(* CODESYS project SimpleFilterPress

Project tree, tasks and I/O mapping:
  CR1082 : CR1082, ifm electronic, order no. PDM360NG, version 3.3.0.2
    application Application
      libraries: VisuDialogs, * (System); CAA Real Time Clock Extern, * (CAA Technical Workgroup); Standard, 3.5.18.0 (System)
      task Task_30ms (cyclic, interval 30 ms, priority 0) calls IO_Block_Organize, POU_MANUAL_CONTROL
      task VISU_TASK (cyclic, interval t#20ms, priority 15) calls VisuElems.Visu_Prg
      GlobalVariables/
        global variables GVL
        global variables GVL_KeyList
        global variables GVL_KeyList_FT
        global variables GVL_KeyList_RT
        global variables GVL_Program_Variables
      image pool ImagePool
      IO Blocks/
        AL1342 Master block/
          program AL1342_IO_Link_Master_A [ST]
        Input Block/
        data type IO_link_port
        Output block/
      Main/
        visualisation Graph
        visualisation Main_Screen
        visualisation Manual
        visualisation Setpoints
        visualisation Stats
      Pressure_Feed/
        program pressure_transducer_1 [ST]: analog_warnings_action
        visualisation W77_1
        visualisation W78_1
        visualisation W79_1
      Pressure_Hydraulic/
        program pressure_transducer [ST]
        visualisation W77
        visualisation W78
        visualisation W79
      PROGRAM_ROUTINES/
        program IO_Block_Organize [CFC]
        program POU_aSeq_Master [LD]
        program POU_MANUAL_CONTROL [LD]
      global variables pVars
      Sentronic/
        program Feed_Diaphram_Pump [ST]
        program POU_Sentronic_ST [ST]
      program SystemTime [ST]
      Warning system/
        function block create_warning [ST]
        Status light/
        program visu_context [ST]
        visualisation W171
        visualisation W172
        visualisation W25
        visualisation W97
        data type warning_message
        global variables warnings_globals
    Communication : Communication, ifm electronic, version 3.3.0.2
      CAN : CAN, ifm electronic, version 3.3.0.2
      Ethernet : Ethernet, ifm electronic, version 3.3.0.2
    Ethernet_1 : Ethernet, CODESYS, version 4.2.0.0
        settings: IPAddress = [192,168,1,247]; SubnetMask = [255,255,255,0]; GatewayAddress = [192,168,1,1]; MACAddress = [16#00,16#02,16#01,16#7B,16#36,16#8D]; NetworkInterfaceName = 'eth0'; NetworkInterfaceName = "eth0"; SaveCommunicationSettings = FALSE
      Modbus_TCP_Master : Modbus TCP Master, 3S - Smart Software Solutions GmbH, version 4.3.0.0
          settings: AutoReconnect = TRUE
    HMI : HMI, ifm electronic, version 3.3.0.2
      Buzzer : Buzzer, ifm electronic, version 3.3.0.2
          output uiBuzzerFreq : UINT  // Frequency
          output xBuzzerON : BIT  // Buzzer ON
      KeyBoards : KeyBoards, ifm electronic, version 3.3.0.2
        Key_Backlight_settings : Key Backlight settings, ifm electronic, version 3.3.0.2
            output xNightModeON : BIT  // Night Mode ON
        Key_Mapping : Key Mapping, ifm electronic, version 3.3.0.2
        Keys : Keys, ifm electronic, version 3.3.0.2
          LEDs_Keyboard_1 : LEDs Keyboard 1, ifm electronic, version 3.3.0.2
              output LEDsKeyboard1 : WORD  // LEDsKeyboard1
          LEDs_Keyboard_3 : LEDs Keyboard 3, ifm electronic, version 3.3.0.2
              output LEDsKeyboard3 : WORD  // LEDs Keyboard 3
      LCD_Backlight : LCD Backlight, ifm electronic, version 3.3.0.2
          output uiBacklightBrightness : UINT  // Brightness
      User_LEDs : User_LEDs, ifm electronic, version 3.3.0.2
          output LED0 : LED_IEC_A_OUTPUT_MAPPING_TYPE  // User LED 0
    Local_IO : Local IO, ifm electronic, version 3.3.0.2
      Inputs : Inputs, ifm electronic, version 3.3.0.2
          input  IN0000 : IN_MULTIFUNCTION_B_INPUT_MAPPING_TYPE  // IN0000
      Outputs : Outputs, ifm electronic, version 3.3.0.2
          output OUT0000 : OUT_DIGITAL_A_OUTPUT_MAPPING_TYPE  // OUT0000
      System_Inputs : System_Inputs, ifm electronic, version 3.3.0.2
          input  uiVoltageVBB30 : UINT  // Voltage VBB30
          input  uiVoltageVBB15 : UINT  // Voltage VBB15
          input  iTemperature0 : INT  // Board Temperature 0
          input  iTemperature1 : INT  // Board Temperature 1
          input  uiLightSensor : UINT  // Light Sensor
    System_Info : System_Info, ifm electronic, version 3.3.0.2
  ecomatDisplay43inch_64bit : ecomatDisplay43inch_64bit, ifm electronic, order no. 
      , version 3.5.19.4
    application Application
      task VISU_TASK (cyclic, interval 100 ms, priority 31) calls VisuElems.Visu_Prg
      GlobalVariables/
      Main_Task/
      Pressure_Feed/
        program pressure_transducer_1 [ST]
        visualisation W77_1
        visualisation W78_1
      Screens/
      Sentronic/
        program Feed_Diaphram_Pump [ST]
        program POU_Sentronic_ST [ST]
    Communication : Communication, ifm electronic, version 3.5.19.4
      CAN : CAN, ifm electronic, version 3.5.19.4
      Ethernet : Ethernet, ifm electronic, version 3.5.19.4
  5ce3da45-db07-42e7-a21c-a00fff4ed8f6|C:\FCW\Full Circle Water\Controls - Documents\Software Versions\graphics\240px-Info_icon_002.svg.png
  5ce3da45-db07-42e7-a21c-a00fff4ed8f6|C:\FCW\Full Circle Water\Controls - Documents\Software Versions\graphics\AL1342.png
  5ce3da45-db07-42e7-a21c-a00fff4ed8f6|C:\FCW\Full Circle Water\Controls - Documents\Software Versions\graphics\AL1342big.jpg
  5ce3da45-db07-42e7-a21c-a00fff4ed8f6|C:\FCW\Full Circle Water\Controls - Documents\Software Versions\graphics\AL1342closeup.png
  5ce3da45-db07-42e7-a21c-a00fff4ed8f6|C:\FCW\Full Circle Water\Controls - Documents\Software Versions\graphics\AL1940.jpg
  5ce3da45-db07-42e7-a21c-a00fff4ed8f6|C:\FCW\Full Circle Water\Controls - Documents\Software Versions\graphics\AL2330.jpg
  5ce3da45-db07-42e7-a21c-a00fff4ed8f6|C:\FCW\Full Circle Water\Controls - Documents\Software Versions\graphics\AL2341.jpg
  5ce3da45-db07-42e7-a21c-a00fff4ed8f6|C:\FCW\Full Circle Water\Controls - Documents\Software Versions\graphics\alert_icon.png
  5ce3da45-db07-42e7-a21c-a00fff4ed8f6|C:\FCW\Full Circle Water\Controls - Documents\Software Versions\graphics\e_stop_button.png
  5ce3da45-db07-42e7-a21c-a00fff4ed8f6|C:\FCW\Full Circle Water\Controls - Documents\Software Versions\graphics\green_check.png
  5ce3da45-db07-42e7-a21c-a00fff4ed8f6|C:\FCW\Full Circle Water\Controls - Documents\Software Versions\graphics\jescochemtanksmall.png
  5ce3da45-db07-42e7-a21c-a00fff4ed8f6|C:\Users\Joe Elvendahl\Pictures\purgepicture.png
  5ce3da45-db07-42e7-a21c-a00fff4ed8f6|C:\Users\Nathan\Full Circle Water\Controls - Documents\Software Versions\graphics\bluebackground 1280x800.png
  5ce3da45-db07-42e7-a21c-a00fff4ed8f6|C:\Users\Nathan\Full Circle Water\Controls - Documents\Software Versions\graphics\FCW1100.png
  5ce3da45-db07-42e7-a21c-a00fff4ed8f6|C:\Users\Nathan\Full Circle Water\Controls - Documents\Software Versions\graphics\FCW720.png
  5ce3da45-db07-42e7-a21c-a00fff4ed8f6|C:\Users\Nathan\Full Circle Water\Controls - Documents\Software Versions\graphics\Stone Phix.png
  5ce3da45-db07-42e7-a21c-a00fff4ed8f6|C:\Users\Nathan\Full Circle Water\Marketing and Sales - Documents\FCW LOGO and BRANDING\Logo\FCW-Logo_Finals\Logo Finals\Full Circle Logo Final-02.png
  5ce3da45-db07-42e7-a21c-a00fff4ed8f6|graphics\AL2240.png
  5ce3da45-db07-42e7-a21c-a00fff4ed8f6|graphics\AL2400.png
  5ce3da45-db07-42e7-a21c-a00fff4ed8f6|graphics\blowdown_valve.png
  5ce3da45-db07-42e7-a21c-a00fff4ed8f6|graphics\bredel_pump.png
  5ce3da45-db07-42e7-a21c-a00fff4ed8f6|graphics\cone.png
  5ce3da45-db07-42e7-a21c-a00fff4ed8f6|graphics\core_blow_valve.png
  5ce3da45-db07-42e7-a21c-a00fff4ed8f6|graphics\doors_closed.png
  5ce3da45-db07-42e7-a21c-a00fff4ed8f6|graphics\doors_open.png
  5ce3da45-db07-42e7-a21c-a00fff4ed8f6|graphics\doors_partly_open.png
  5ce3da45-db07-42e7-a21c-a00fff4ed8f6|graphics\head_valves.png
  5ce3da45-db07-42e7-a21c-a00fff4ed8f6|graphics\hydraulic_pressure_sensor.png
  5ce3da45-db07-42e7-a21c-a00fff4ed8f6|graphics\hydraulic_pump_contactor.png
  5ce3da45-db07-42e7-a21c-a00fff4ed8f6|graphics\hydraulic_temp_and_level.png
  5ce3da45-db07-42e7-a21c-a00fff4ed8f6|graphics\membrane_squeeze_contactor.png
  5ce3da45-db07-42e7-a21c-a00fff4ed8f6|graphics\metal_aro_pump.jpg
  5ce3da45-db07-42e7-a21c-a00fff4ed8f6|graphics\mixer.png
  5ce3da45-db07-42e7-a21c-a00fff4ed8f6|graphics\plate_shifter.png
  5ce3da45-db07-42e7-a21c-a00fff4ed8f6|graphics\press_open.png
  5ce3da45-db07-42e7-a21c-a00fff4ed8f6|graphics\press_side_view.png
  5ce3da45-db07-42e7-a21c-a00fff4ed8f6|graphics\R08_andR09_masters.jpg
  5ce3da45-db07-42e7-a21c-a00fff4ed8f6|graphics\radar_pod.png
  5ce3da45-db07-42e7-a21c-a00fff4ed8f6|graphics\servo_drives.png
  5ce3da45-db07-42e7-a21c-a00fff4ed8f6|graphics\single_filter_plate.png
  5ce3da45-db07-42e7-a21c-a00fff4ed8f6|graphics\squeeze_transducer.png
  5ce3da45-db07-42e7-a21c-a00fff4ed8f6|graphics\squeeze_valve.png
  5ce3da45-db07-42e7-a21c-a00fff4ed8f6|graphics\vector_hose_pump.jpg
  5ce3da45-db07-42e7-a21c-a00fff4ed8f6|graphics\wet_end_master.png
  text list GlobalTextList
*)

// CR1082/Application/IO Blocks/IO_link_port
TYPE IO_link_port :
	STRUCT 
		vendor_ID: UINT;						//  The vendor ID reported by an IO-Link device.
		device_ID: UINT;						//  The model ID number reported by an IO-Link device.
		
		port_ID: STRING;					//  A text description of the port, ie. 'X.02'.   Used for warning visus, such as 'short circuit on port xx'
		port_number: INT;					//  The simple port number.   Used by modbus libraries to directly read/write if they choose to do so.
		block_name: STRING;					//  The name of the device, ie. 'AL1342'.  Used by visus to describe where something is connected, but also by the modbus libraries for direct reads/writes.
		
		DI_pin_4: BOOL;						//  Digital input #1 (pin 4), if port is configured as an input.
		DI_pin_2: BOOL;						//  Digital input #2 (pin 2).   This pin works if the port is configured as IO-Link or as an input.
		
		not_connected: BOOL;				//  Nothing is connected to the port (only works in IO-Link mode.)
		data_invalid: BOOL;					//  Something is connected but it's not communicating correctly (only works in IO-Link mode.)
		
		short_circuit: BOOL;				//  The device on this port has drawn more current than the port can provide.  (300 mA on an AL1342.)
		
		master_disconnected: BOOL;			//  The master block itself isn't connected, so we should ignore individual device disconnections.
		
		read_word_0: WORD;					//  Process data word 0
		read_word_1: WORD;					//  Process data word 1
		read_word_2: WORD;					//  Process data word 2
		read_word_3: WORD;					//  Process data word 3
		read_word_4: WORD;					//  Process data word 4
		read_word_5: WORD;					//  Process data word 5
		read_word_6: WORD;					//  Process data word 6

		write_word_0: WORD;					//  Write to device word 0
		write_word_1: WORD;					//  Write to device word 1
		write_word_2: WORD;					//  Write to device word 2
		write_word_3: WORD;					//  Write to device word 3
		
		DO_pin_4: BOOL;						//  Set pin 4 to on or off (if the IO-Link port is configured as an output.)
		
	END_STRUCT
END_TYPE

// CR1082/Application/Warning system/warning_message
TYPE warning_message :
	STRUCT 
		detail_warning_visu: STRING := ''; 		//  The exact name of the associated warning visualization.  The warning system uses this string to match visualizations and to match duplicate or fixed messages.
		red: BOOL := FALSE;    					//  Is it a 'red' warning?  (System needs immediate attention.)
		yellow: BOOL := FALSE;   				//  Is it a 'yellow'? warning?  (System needs attention eventually.)
		fixed: BOOL := FALSE;    				//  Has the problem been fixed?
		informational: BOOL := FALSE; 			//  Is this just a general message, not a fault?
		pop_up_everywhere: BOOL := FALSE;  		//  Set if we should immediately switch to the detail warning screen no matter what (high priority.)
		pop_up_contextual: BOOL := FALSE;  		//  Set if we should switch to warning detail screen when they enter the corresponding section of the interface, ie. a VFD fault pops when they go to Return Pump
		contextual_visu: STRING := '';  		//  the visualization we should pop up the warning on.
		short_Description: STRING;   			//  This is the description that will appear in the Warning log.
		audible_alarm: BOOL;     				//  If checked, I suggest adding a 'silence alarm' button to the corresponding Warning visu that sets GVL.siren := FALSE;  Siren automatically silences when you go to a Warnings screen
		time_stamp:	DATE_AND_TIME;   			//  The warning automatically gets time stamped; you never need to set this.
		fixed_date_time: DATE_AND_TIME;			//  When was the message marked as fixed?  Also automatically time-stamped.
		truncated_code: INT;					//  Used to reduce the visualization name to an integer that can be easily passed through say a modbus register.  Automatically generated.
	END_STRUCT
END_TYPE

//  To use these Warning messages, they are either passed to the Warnings() function directly, or assigned to an instance of the create_warning function block (which then sends it as needed
//  to the Warnings() function.)

//  The minimum required fields for a Warning message are:   short_Description, detail_warning_visu, and one of the 'type' flags (red, yellow, fixed, or informational.)
//  Everything else is optional.   Time stamping happens automatically.

//  The tradition (but not requirement) is to set the pop_up_everywhere flag to TRUE for 'red' warnings.

//  Example of a minimal complete Warning message:

//  shorted_port_message: warning := (red := TRUE, detail_warning_visu := 'W276', short_Description := 'Shorted output block port');

// CR1082/Application/pVars
{attribute 'qualified_only'}
VAR_GLOBAL PERSISTENT RETAIN

	run: BOOL; 			// The master enable switch for the system, tied to the button in the upper left corner of the main screen.

	
//  System options

	screen_brightness : USINT := 70; 	// 0-100% screen brightness
	use_metric_units : BOOL; 			// If true, display metric units of measurement
	user_pin: INT := 12345; 			// The system pin number.
	relock_after_x_minutes: TIME:= T#10M;	//  How long should a login with the PIN be good for?
	require_pin_to_change_setting: BOOL := FALSE;
	require_pin_to_start : BOOL := FALSE;
	
	power_restored_time: DATE_AND_TIME;				// The time the system last booted up
	power_lost: DATE_AND_TIME;						// The time we lost power at.
	we_had_power_now: DATE_AND_TIME;				// Tracks the time of the most recent execution of the Status_Light program.

//   Clarifier

gallons_since_last_purge: REAL;
purge_frequency_gallons: INT := 3000;
purge_duration: TIME := T#15S;


//   Flow meter

flow_sensor_pipe_cross_section: REAL;				// The cross section (in square inches) of the pipe the thermal mass flow sensor (SM8621) is installed in.

//  Chemical system

analog_coagulant_sensor_installed: BOOL;			// TRUE if we are using an IO-Link analog level sensor on the coagulant tank.
coagulant_tank_empty_level_inches: INT;				//
coagulant_tank_gallons_per_inch: REAL;				//
coagulant_tank_low_level_warning_inches: INT;		//

analog_floc_concentrate_sensor_installed: BOOL;		// TRUE if we are using an IO-Link analog level sensor on the flocculant concentrate tank.
floc_concentrate_empty_level_inches: INT;
floc_conc_gallons_per_inch: REAL;
floc_conc_low_level_warning_inches: INT;

diluted_floc_analog_sensor_installed: BOOL;			// TRUE if we are using an IO-Link analog level sensor on the flocculant concentrate tank.
diluted_floc_empty_level_inches: INT;
diluted_floc_gallons_per_inch: REAL;
diluted_floc_low_level_warning_inches: INT;

//  Mechanical pit mixer

	mechanical_mixer_installed: BOOL;			//  True if the system has a mechanical pit mixer
	Feed_Diaphram_Pump_Enabled: BOOL;				//  True if the mechanical pit mixer is enabled
	Feed_Pump_Speed: REAL;				//  A percentage speed (100 = max speed, or 60 Hz.)

//  Warning system

	myWarnings: ARRAY [1..16] OF warning_message;
	redWarningPresent: BOOL;					// TRUE if there's an active red (critical) warning
	yellowWarningPresent: BOOL;					// TRUE if there's an active yellow (caution/attention) warning
	blueWarningPresent: BOOL;					// TRUE if there's an active blue (informational) warning
	warningButtonLights: INT;					// Used by the old CR1082 controller to turn on/off button lights for the Warnings screen
	
	slave_trip_code: INT;						// The last fault code generated by the slave plate shifter servo
	master_trip_code: INT;						// The last fault code generated by the master plate shifter servo

	last_warning_number: int;					//  The numerical portion of the warning short code, ie. W-201 becomes '201'.
	
// Water tank
	max_level_inches: REAL := 65;		
	low_level_percent: REAL;
	out_of_water_level_percent: REAL;
	
	// Filter Press Setpoints
		Hydraulic_PSI_Setpoint: REAL;
		Air_Blow_Minutes: REAL;
		Cake_Feed_PSI_Setpoint: REAL;
		Cake_Feed_Time_Delay_Secs: REAL;
		Cake_Stepup_Factor: REAL;
		Sentronic_Word: WORD;
		Sentronic_Real: REAL;
		
		
	
	
//  Pressure transducer

	pressure_transducer_type: INT;			//  The deviceID of the last known pressure transducer we saw from the 'pressure_transducer' program.
	


END_VAR

// CR1082/Application/GlobalVariables/GVL
{attribute 'qualified_only'}
VAR_GLOBAL
	

	runGreenHalo: BOOL := FALSE;  // shows (FALSE) or hides (TRUE) the green 'RUNNING' ring around the RUN/STOP button on the main screen.
	phYellowHalo: BOOL := FALSE;  // TRUE to show a yellow (minor fault) halo around the "pH Control" button on the main screen when there is a minor problem with the pH system
	phRedHalo: BOOL := FALSE;	  // TRUE to show a red (critical fault) halo around the "pH Control" button on the main screen when there is a serious problem with the pH system
	sanitizerYellowHalo: BOOL := TRUE;  // FALSE to show a yellow (minor fault) halo around the "Sanitizer" button on the main screen when there is a minor problem with the bromine system
	sanitizerRedHalo: BOOL := TRUE;     // FALSE to show a red (critical fault) halo around the "Sanitizer" button on the main screen when there is a serious problem with the bromine system

	show_change_time: BOOL;			// True if we want to display the frame to change the time settings.
	
	WarningButtonPressed: INT;    // this tells the Warning system which button was pressed on the Warning Log screen
	WarningGlobalReset: BOOL := FALSE;   //  The reset button on the Warning Log screen toggles this to true, which signals Warnings (PRG)
	warningSecondaryReset: BOOL := FALSE;  //  This is the signal to the rest of the system to re-set all 'warning sent' flags.
	resettime: TIME;   //   When the initial warning reset button was pressed, lets the Warnings PRG decide when to stop broadcasting the reset signal.
	forcekeylightupdate: BOOL;  // gives us an extra way to trigger the update mechanism for key lights without actually changing the visu
	siren: BOOL;   // Master switch to turn the audible siren of the stack light on and off.
	
	

END_VAR

// CR1082/Application/GlobalVariables/GVL_KeyList
{attribute 'qualified_only'}

(* 

!!! This GVL list is from project template !!!

The following variables are controlled by key events mapped at Default Hotkey mapping list in Visualization Manager.

For example, F1 function key of standard keyboard (MFII) is pressed, xF1 bit in this list will become TRUE; when the same 
key is released then xF1 become FALSE.

*)

VAR_GLOBAL

(* Display system key press / release event status. TRUE = Key Pressed, FALSE = Key Released  *)
	xF1 		: BOOL;		(* Event status of F1 function key *)
	xF2 		: BOOL;		(* Event status of F2 function key *)
	xF3 		: BOOL;		(* Event status of F3 function key *)
	xF4 		: BOOL;		(* Event status of F4 function key *)
	xF5 		: BOOL;		(* Event status of F5 function key *)
	xF6 		: BOOL;		(* Event status of F6 function key *)
	xF7 		: BOOL;		(* Event status of F7 function key *)
	xF8 		: BOOL;		(* Event status of F8 function key *)
	xF9 		: BOOL;		(* Event status of F9 function key *)
	xF10 		: BOOL;		(* Event status of F10 function key *)
	xUp 		: BOOL;		(* Event status of Up arrow key *)
	xDown		: BOOL;		(* Event status of Down arrow key *)
	xLeft 		: BOOL;		(* Event status of Left arrow key *)
	xRight 		: BOOL;		(* Event status of Right arrow key *)
	xKey_Return : BOOL;		(* Event status of Return (or Enter) key *)
END_VAR

// CR1082/Application/GlobalVariables/GVL_KeyList_FT
{attribute 'qualified_only'}

(* 

!!! This GVL list is from project template !!!

The following variables returns a pulse for one scan cycle when a respective key is released (i.e. at falling trigger).
These key release event is detected by the state of variables in GVL GVL_KeyList.

For example, F1 function key of standard keyboard (MFII) is released, xF1 bit in this list will become TRUE for one scan cycle.

*)

VAR_GLOBAL

(* Display system key release event falling trigger pulse. *)
	xF1 		: BOOL;		(* Event status of F1 function key *)
	xF2 		: BOOL;		(* Event status of F2 function key *)
	xF3 		: BOOL;		(* Event status of F3 function key *)
	xF4 		: BOOL;		(* Event status of F4 function key *)
	xF5 		: BOOL;		(* Event status of F5 function key *)
	xF6 		: BOOL;		(* Event status of F6 function key *)
	xF7 		: BOOL;		(* Event status of F7 function key *)
	xF8 		: BOOL;		(* Event status of F8 function key *)
	xF9 		: BOOL;		(* Event status of F9 function key *)
	xF10 		: BOOL;		(* Event status of F10 function key *)
	xUp 		: BOOL;		(* Event status of Up arrow key *)
	xDown		: BOOL;		(* Event status of Down arrow key *)
	xLeft 		: BOOL;		(* Event status of Left arrow key *)
	xRight 		: BOOL;		(* Event status of Right arrow key *)
	xKey_Return : BOOL;		(* Event status of Return (or Enter) key *)
END_VAR

// CR1082/Application/GlobalVariables/GVL_KeyList_RT
{attribute 'qualified_only'}

(* 

!!! This GVL list is from project template !!!

The following variables returns a pulse for one scan cycle when a respective key is pressed (i.e. at rising trigger)
These key press event is detected by the state of variables in GVL GVL_KeyList.

For example, F1 function key of standard keyboard (MFII) is pressed, xF1 bit in this list will become TRUE for one scan cycle.

*)

VAR_GLOBAL

(*Display system key press event rising trigger pulse *)
	xF1 		: BOOL;		(* Event status of F1 function key *)
	xF2 		: BOOL;		(* Event status of F2 function key *)
	xF3 		: BOOL;		(* Event status of F3 function key *)
	xF4 		: BOOL;		(* Event status of F4 function key *)
	xF5 		: BOOL;		(* Event status of F5 function key *)
	xF6 		: BOOL;		(* Event status of F6 function key *)
	xF7 		: BOOL;		(* Event status of F7 function key *)
	xF8 		: BOOL;		(* Event status of F8 function key *)
	xF9 		: BOOL;		(* Event status of F9 function key *)
	xF10 		: BOOL;		(* Event status of F10 function key *)
	xUp 		: BOOL;		(* Event status of Up arrow key *)
	xDown		: BOOL;		(* Event status of Down arrow key *)
	xLeft 		: BOOL;		(* Event status of Left arrow key *)
	xRight 		: BOOL;		(* Event status of Right arrow key *)
	xKey_Return : BOOL;		(* Event status of Return (or Enter) key *)
END_VAR

// CR1082/Application/GlobalVariables/GVL_Program_Variables
{attribute 'qualified_only'}
VAR_GLOBAL
	GVL_START_PB: BOOL;
	GVL_STOP_PB: BOOL;
	GVL_START_IND: BOOL;
	GVL_MACHINE_RUNNING: BOOL;
	GVL_SEQ_MASTER: INT;
	GVL_SEQ_FEED: INT;
	GVL_SEQ_HYD: INT;
	GVL_HYD_PSI: REAL;
	GVL_FEED_PSI: REAL;
	GVL_DISPLAY_TIME: REAL;
	GVL_CAKE_ET: TIME;
	GVL_AIRBLOW_ET: TIME;
	GVL_DISPLAY_SETPOINT: REAL;
	GVL_DISPLAY_TIME_SP: TIME;
	GVL_DISPLAY_TIME_ET: TIME;
	GVL_AIRBLOW_SOLENOID: BOOL;
	GVL_LAST_CYCLE_TIME: REAL;
	GVL_CAKE_ET_REAL: REAL;
	GVL_CAKE_SETPOINT_TIME: TIME;
	GVL_AIRBLOW_MIN_TIME: TIME;
	GVL_CAKE_CYCLE_TIME: TIME;
	GVL_CAKE_CYCLE_ACC: TIME;
	GVL_FULL_CYCLE_TIME: TIME;
	GVL_MAN_AIR_BLOW_PB: BOOL;
	GVL_MAN_AIR_BLOW_BIT: BOOL;
	GVL_MAN_DIAPHRAM_PUMP: BOOL;
	
	
	
	
	
	
END_VAR

// CR1082/Application/Warning system/warnings_globals
{attribute 'qualified_only'}
VAR_GLOBAL
	last_pop_up_time: TIME;
		
	WarningButtonPressed: INT;   		 	//  This tells the Warning system which button was pressed on the Warning Log screen, ie. button 1 = myWarnings[1]
	warning_screen: INT := 1;				//  Which of the Warning log screens did we last come from?  1 = warning_log, 2 = warning_log_2
	WarningGlobalReset: BOOL := FALSE;   	//  The reset button on the Warning Log screen toggles this to true, which signals Warnings (PRG)
	warningSecondaryReset: BOOL := FALSE;  	//  This is the signal to the rest of the system to re-set all 'warning sent' flags.
	resettime: TIME;   //   When the initial warning reset button was pressed, lets the Warnings PRG decide when to stop broadcasting the reset signal.
	update_status_light: BOOL;  // gives us an extra way to trigger the update mechanism for key lights without actually changing the visu
	siren: BOOL;   // Master switch to turn the audible siren of the stack light on and off.
	in_setup: BOOL;							//  If TRUE, suppress pop-up warnings.  This keeps the system from interrupting during the configuration process.
END_VAR

// CR1082/Application/PROGRAM_ROUTINES/IO_Block_Organize
PROGRAM IO_Block_Organize
VAR
END_VAR
VAR // added by the converter: edge detectors and wires of the graphical bodies
    _w1, _w2 : REAL;
END_VAR

POU_ASEQ_MASTER();
AL1342_IO_LINK_MASTER_A();
PRESSURE_TRANSDUCER_1(IO_Link_port := AL1342_IO_LINK_MASTER_A.X_03);
PRESSURE_TRANSDUCER(IO_Link_port := AL1342_IO_LINK_MASTER_A.X_01);
_w1 := TO_REAL(GVL_Program_Variables.GVL_DISPLAY_TIME_ET) * 0.001;
_w2 := TO_REAL(GVL_Program_Variables.GVL_DISPLAY_TIME_SP) * 0.001;
GVL_Program_Variables.GVL_CAKE_ET_REAL := TO_REAL(GVL_Program_Variables.GVL_CAKE_ET) * 0.001;
GVL_Program_Variables.GVL_AIRBLOW_MIN_TIME := TO_TIME(PVARS.Air_Blow_Minutes);
GVL_Program_Variables.GVL_DISPLAY_TIME := _w1;
GVL_Program_Variables.GVL_DISPLAY_SETPOINT := _w2;
GVL_Program_Variables.GVL_CAKE_SETPOINT_TIME := TO_TIME(pVars.Cake_Feed_Time_Delay_Secs);
OUTPUT_BLOCK(x1_0_pin4 := GVL_Program_Variables.GVL_AIRBLOW_SOLENOID, IO_Link_port := AL1342_IO_LINK_MASTER_A.X_08);
Feed_Diaphram_Pump(Sentronic_Real := POU_ASEQ_MASTER.Sentronic_Command, DP1213_IO_link := AL1342_IO_LINK_MASTER_A.X_05);

END_PROGRAM

// CR1082/Application/PROGRAM_ROUTINES/POU_aSeq_Master
PROGRAM POU_aSeq_Master
VAR
	Hyd_Low_PSI_Shutoff: REAL;
	TON_0: TON;
	temp_real: REAL;
	
	temp: REAL;	
	
	
	
	TON_0_ETIMe: real;
	Message_String: string;
	temp_2: REAL;
	TON_1: TON;
	Air_Blow_Time: real;
	Display_Time: real;
	TON_2: TON;
	TEMP_TIME: TIME;
	temp_5: INT;
	TEMP_SOLENOID: BOOL;
END_VAR

VAR_OUTPUT
	Sentronic_Command: REAL;
END_VAR
VAR // added by the converter: edge detectors and wires of the graphical bodies
    _w1, _w2, _w3, _w4, _w5, _w6, _w7, _w8 : BOOL;
END_VAR

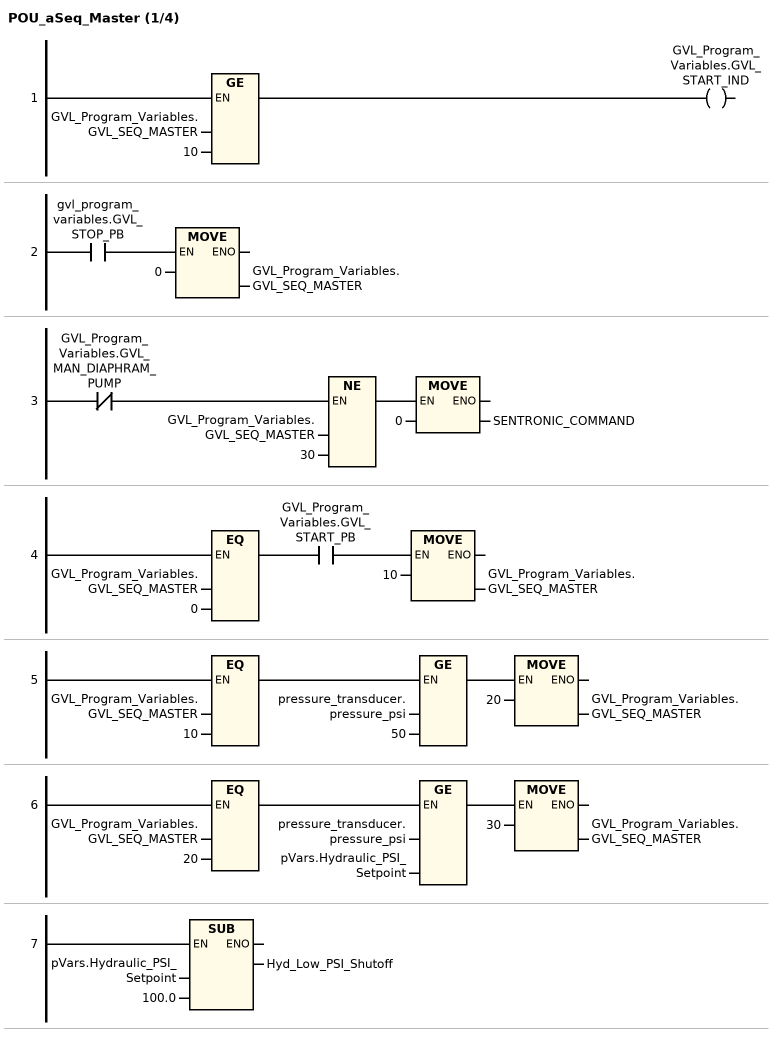
// NETWORK 1
GVL_Program_Variables.GVL_START_IND := GVL_Program_Variables.GVL_SEQ_MASTER >= 10;

// NETWORK 2
IF gvl_program_variables.GVL_STOP_PB THEN GVL_Program_Variables.GVL_SEQ_MASTER := 0; END_IF

// NETWORK 3
IF NOT GVL_Program_Variables.GVL_MAN_DIAPHRAM_PUMP AND GVL_Program_Variables.GVL_SEQ_MASTER <> 30 THEN
    SENTRONIC_COMMAND := 0;
END_IF

// NETWORK 4
IF GVL_Program_Variables.GVL_SEQ_MASTER = 0 AND GVL_Program_Variables.GVL_START_PB THEN
    GVL_Program_Variables.GVL_SEQ_MASTER := 10;
END_IF

// NETWORK 5
IF GVL_Program_Variables.GVL_SEQ_MASTER = 10 AND pressure_transducer.pressure_psi >= 50 THEN
    GVL_Program_Variables.GVL_SEQ_MASTER := 20;
END_IF

// NETWORK 6
IF GVL_Program_Variables.GVL_SEQ_MASTER = 20 AND pressure_transducer.pressure_psi >= pVars.Hydraulic_PSI_Setpoint THEN
    GVL_Program_Variables.GVL_SEQ_MASTER := 30;
END_IF

// NETWORK 7
Hyd_Low_PSI_Shutoff := pVars.Hydraulic_PSI_Setpoint - 100.0;

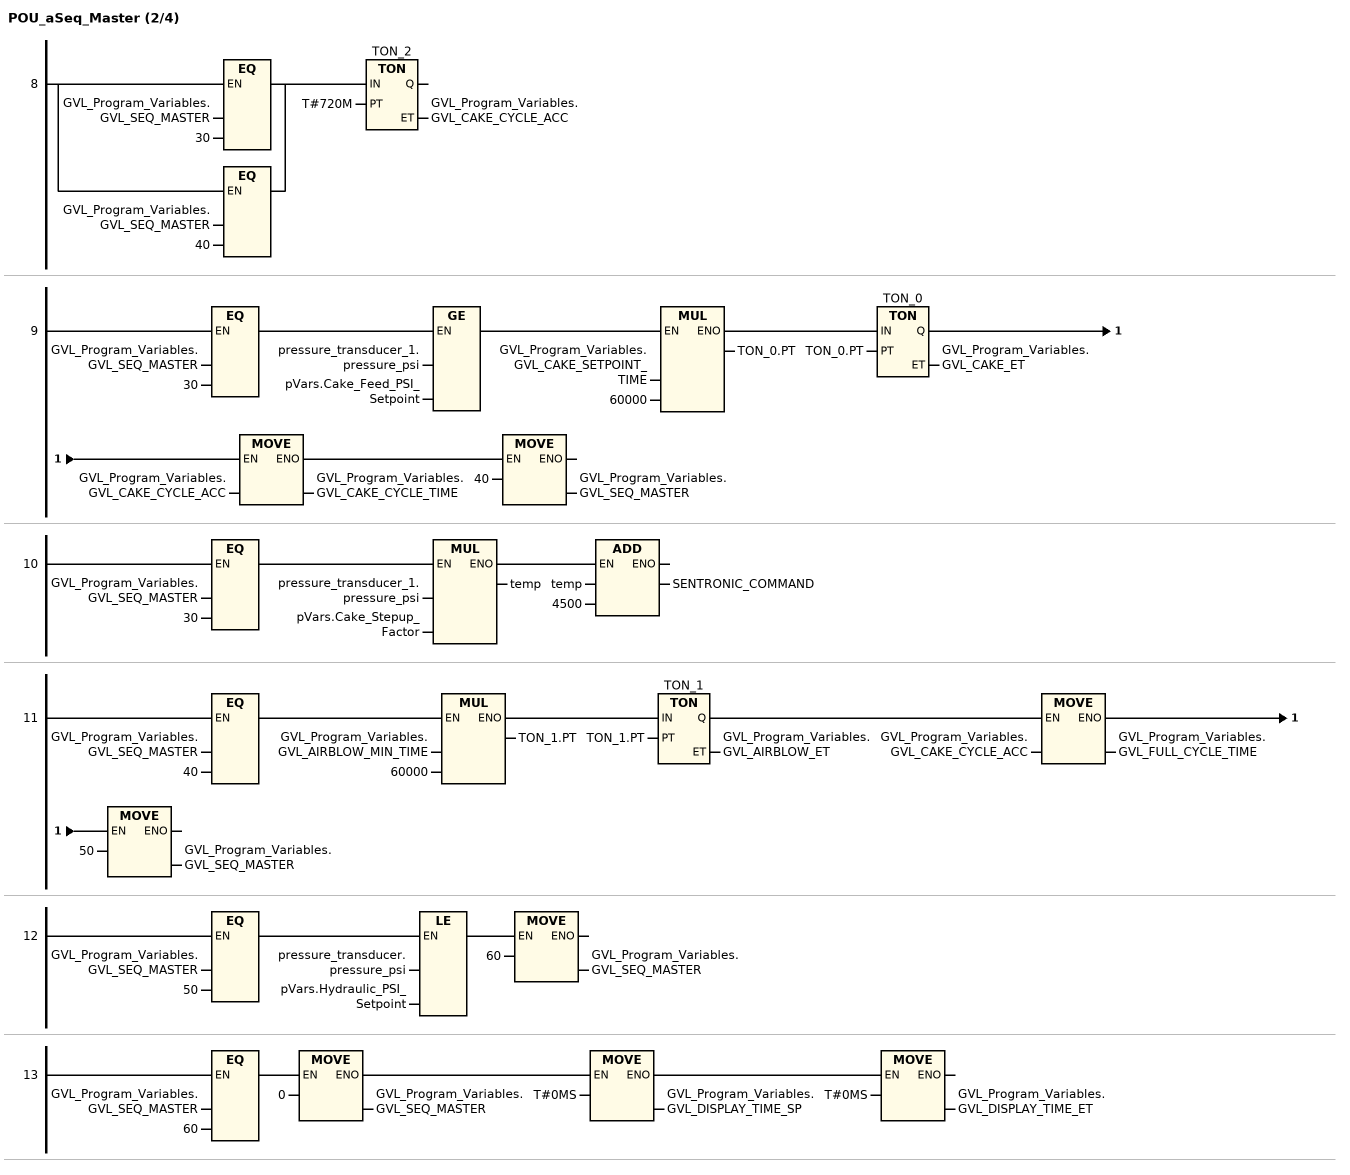
// NETWORK 8
TON_2(
    IN := GVL_Program_Variables.GVL_SEQ_MASTER = 30 OR GVL_Program_Variables.GVL_SEQ_MASTER = 40,
    PT := T#720M,
    ET => GVL_Program_Variables.GVL_CAKE_CYCLE_ACC); // TON

// NETWORK 9
_w1 := GVL_Program_Variables.GVL_SEQ_MASTER = 30 AND pressure_transducer_1.pressure_psi >= pVars.Cake_Feed_PSI_Setpoint;
IF _w1 THEN TON_0.PT := GVL_Program_Variables.GVL_CAKE_SETPOINT_TIME * 60000; END_IF
TON_0(IN := _w1, PT := TON_0.PT, ET => GVL_Program_Variables.GVL_CAKE_ET); // TON
_w2 := TON_0.Q;
IF _w2 THEN GVL_Program_Variables.GVL_CAKE_CYCLE_TIME := GVL_Program_Variables.GVL_CAKE_CYCLE_ACC; END_IF
IF _w2 THEN GVL_Program_Variables.GVL_SEQ_MASTER := 40; END_IF

// NETWORK 10
_w3 := GVL_Program_Variables.GVL_SEQ_MASTER = 30;
IF _w3 THEN temp := pressure_transducer_1.pressure_psi * pVars.Cake_Stepup_Factor; END_IF
IF _w3 THEN SENTRONIC_COMMAND := temp + 4500; END_IF

// NETWORK 11
_w4 := GVL_Program_Variables.GVL_SEQ_MASTER = 40;
IF _w4 THEN TON_1.PT := GVL_Program_Variables.GVL_AIRBLOW_MIN_TIME * 60000; END_IF
TON_1(IN := _w4, PT := TON_1.PT, ET => GVL_Program_Variables.GVL_AIRBLOW_ET); // TON
_w5 := TON_1.Q;
IF _w5 THEN GVL_Program_Variables.GVL_FULL_CYCLE_TIME := GVL_Program_Variables.GVL_CAKE_CYCLE_ACC; END_IF
IF _w5 THEN GVL_Program_Variables.GVL_SEQ_MASTER := 50; END_IF

// NETWORK 12
IF GVL_Program_Variables.GVL_SEQ_MASTER = 50 AND pressure_transducer.pressure_psi <= pVars.Hydraulic_PSI_Setpoint THEN
    GVL_Program_Variables.GVL_SEQ_MASTER := 60;
END_IF

// NETWORK 13
_w6 := GVL_Program_Variables.GVL_SEQ_MASTER = 60;
IF _w6 THEN GVL_Program_Variables.GVL_SEQ_MASTER := 0; END_IF
IF _w6 THEN GVL_Program_Variables.GVL_DISPLAY_TIME_SP := T#0MS; END_IF
IF _w6 THEN GVL_Program_Variables.GVL_DISPLAY_TIME_ET := T#0MS; END_IF

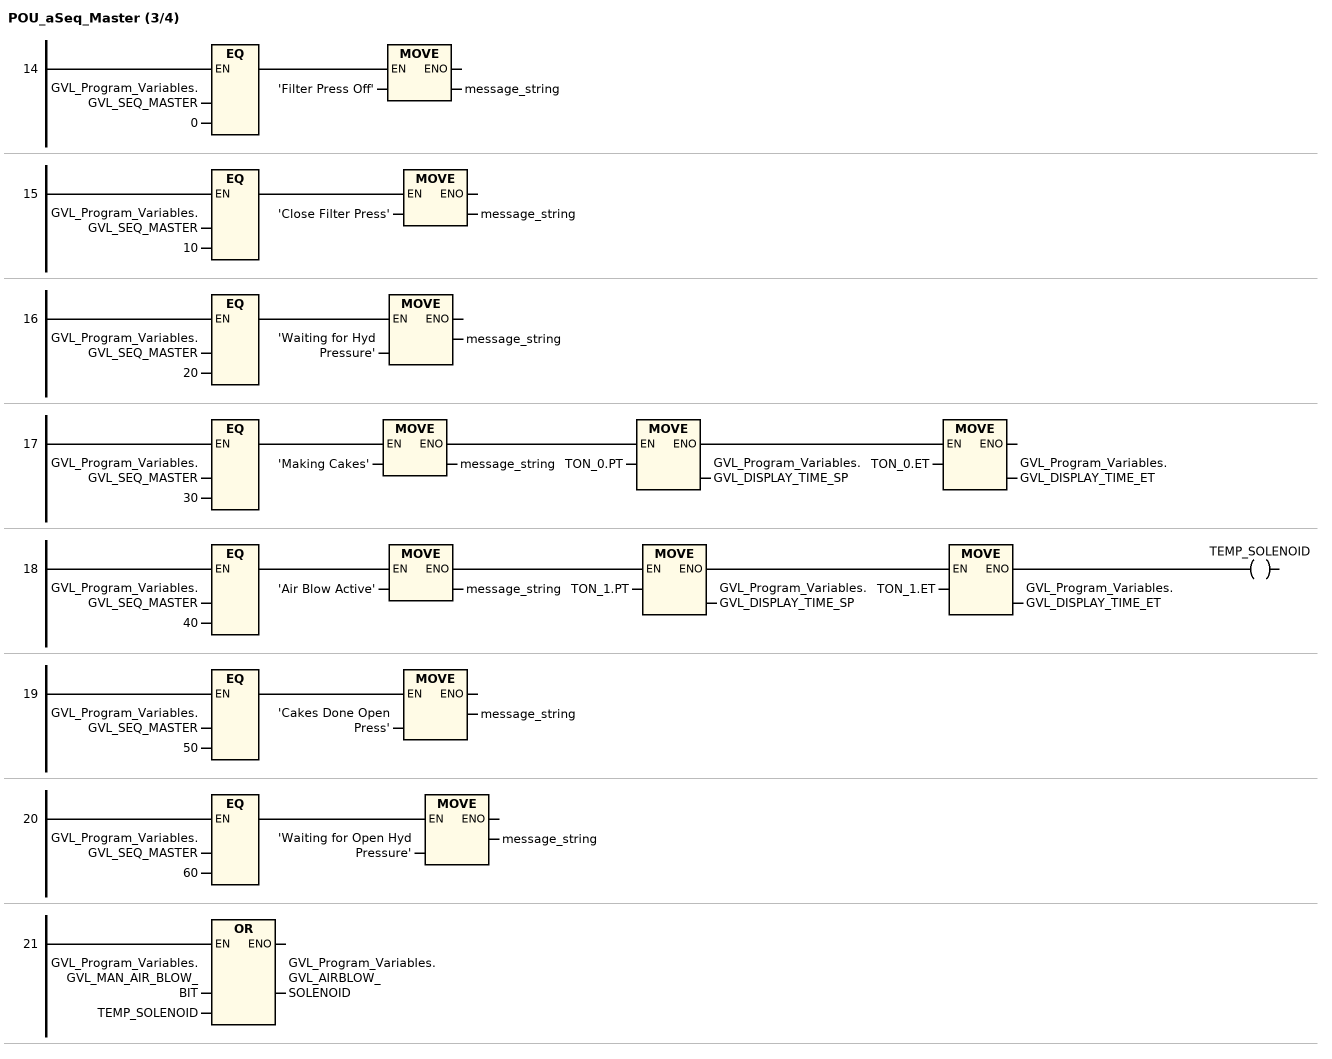
// NETWORK 14
IF GVL_Program_Variables.GVL_SEQ_MASTER = 0 THEN message_string := 'Filter Press Off'; END_IF

// NETWORK 15
IF GVL_Program_Variables.GVL_SEQ_MASTER = 10 THEN message_string := 'Close Filter Press'; END_IF

// NETWORK 16
IF GVL_Program_Variables.GVL_SEQ_MASTER = 20 THEN message_string := 'Waiting for Hyd Pressure'; END_IF

// NETWORK 17
_w7 := GVL_Program_Variables.GVL_SEQ_MASTER = 30;
IF _w7 THEN message_string := 'Making Cakes'; END_IF
IF _w7 THEN GVL_Program_Variables.GVL_DISPLAY_TIME_SP := TON_0.PT; END_IF
IF _w7 THEN GVL_Program_Variables.GVL_DISPLAY_TIME_ET := TON_0.ET; END_IF

// NETWORK 18
_w8 := GVL_Program_Variables.GVL_SEQ_MASTER = 40;
IF _w8 THEN message_string := 'Air Blow Active'; END_IF
IF _w8 THEN GVL_Program_Variables.GVL_DISPLAY_TIME_SP := TON_1.PT; END_IF
IF _w8 THEN GVL_Program_Variables.GVL_DISPLAY_TIME_ET := TON_1.ET; END_IF
TEMP_SOLENOID := _w8;

// NETWORK 19
IF GVL_Program_Variables.GVL_SEQ_MASTER = 50 THEN message_string := 'Cakes Done Open Press'; END_IF

// NETWORK 20
IF GVL_Program_Variables.GVL_SEQ_MASTER = 60 THEN message_string := 'Waiting for Open Hyd Pressure'; END_IF

// NETWORK 21
GVL_Program_Variables.GVL_AIRBLOW_SOLENOID := GVL_Program_Variables.GVL_MAN_AIR_BLOW_BIT OR TEMP_SOLENOID;

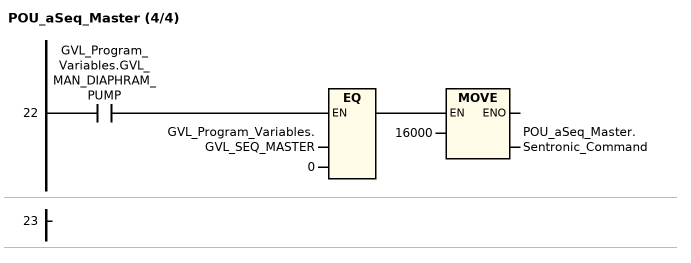
// NETWORK 22
IF GVL_Program_Variables.GVL_MAN_DIAPHRAM_PUMP AND GVL_Program_Variables.GVL_SEQ_MASTER = 0 THEN
    POU_aSeq_Master.Sentronic_Command := 16000;
END_IF

// NETWORK 23

END_PROGRAM

// CR1082/Application/Pressure_Hydraulic/pressure_transducer
//   This program is designed to support a variety of IO-Link pressure transducers.
//   Currently supported:
//		-IFM PM1707 pressure transducer.    https://www.ifm.com/us/en/product/PM1707    Add more sensors if you like.  :-)
//		-IFM PM1789 pressure transducer. 
//		-IFM PV7600 pressure transducer. 
//		-IFM PV7601 pressure transducer. 
//		-IFM PV7602 pressure transducer. 
//		-IFM PV7603 pressure transducer. 	
//		-IFM PV7604 pressure transducer. 


PROGRAM pressure_transducer
VAR
	startup_loop_ran: BOOL;		//  We have completed our startup check for the type of level sensor.

	//   WARNINGS
	
	//  Unknown sensor Warning
	
	unknown_sensor_message: warning_message := (red := TRUE, pop_up_everywhere := TRUE, detail_warning_visu := 'W79', short_Description := 'Unknown pressure transducer');
	unknown_sensor_warning: create_warning;

	//  Disconnected sensor Warning

	disconnected_sensor_message: warning_message := (red := TRUE, pop_up_everywhere := TRUE, detail_warning_visu := 'W77', short_Description := 'Pressure transducer disconnected');
	disconnected_sensor_warning: create_warning;

	//  Shorted sensor Warning
		
	shorted_sensor_message: warning_message := (red := TRUE, pop_up_everywhere := TRUE, detail_warning_visu := 'W78', short_Description := 'Pressure transducer shorted');
	shorted_sensor_warning: create_warning;


END_VAR

VAR_INPUT
END_VAR

VAR_OUTPUT
	pressure_psi: REAL;				//  The current pressure in pounds per square inch
	water_depth_inches: REAL;		//  The depth of water needed to produce this pressure
	temperature_F: real;			//  Temp in degrees F, not available for most sensors.
END_VAR

VAR_IN_OUT
	IO_Link_port: IO_link_port;				// Connect to an IO_link read port.   Used to communicate with an analog level sensor, if so equipped.
END_VAR

IF NOT startup_loop_ran THEN pressure_transducer.startup_loop(); END_IF			//  This startup loop looks for and identifies what kind of sensor we have available.

analog_warnings_action();   			//  Check all the Warnings associated with these pressure sensors


//   Interpret our data according to the type of sensor:

CASE IO_Link_port.device_ID OF
//	668:  pressure_psi := IO_Link_port.read_word_0 * 0.0014504;			//  PM1707.  Native reading is in tenths of a millibar, this converts to psi.

	851:  pressure_psi := IO_Link_port.read_word_0 * 1.4504 ;			//  PV7600.  Native reading is in tenths of a bar, this converts to psi.

//	852:  pressure_psi := IO_Link_port.read_word_0 * 1.4504;			//  PV7601.  Native reading is in tenths of a bar, this converts to psi.
	
//	853:  pressure_psi := IO_Link_port.read_word_0 * 0.14504 ;			//  PV7602.  Native reading is in hundredths of a bar, this converts to psi.
	
//	854:  pressure_psi := IO_Link_port.read_word_0 * 0.14504;			//  PV7603.  Native reading is in hundredths of a bar, this converts to psi.
	
//	855:  pressure_psi := IO_Link_port.read_word_0 * 0.014504;			//  PV7604.  Native reading is in thousandths of a bar, this converts to psi.
	
//   1436:  pressure_psi := IO_Link_port.read_word_0 * 0.00145;			//  PL1506.  Native reading is in tenths of a millibar, this converts to psi.
		  temperature_F := IO_Link_port.read_word_2 * 0.018 + 32;		//  Native reading is in hundredths of a degree C, this converts to F.
		  
		  
		  
	  
		//  New sensors can be added here.  Warning code must be updated if you add (for the 'unknown sensor' Warning)
END_CASE

END_PROGRAM

// CR1082/Application/Warning system/create_warning
//  This function block takes care of some of the drudgery of sending and managing Warning messages.   It has a built-in timer (if you don't want your Warning to trigger
//  immediately), resets Warnings if the user hits the RESET button on the Warning screen, automatically generates 'fixed' messages (derived from your original Warning
//  message) and sends that 'fixed' message if the fault condition no longer exists.
//  It also automatically re-synchronizes warnings with the master Warnings list after a reboot or loss of power (so no persistent variables are needed.)

//  Last modified:  2/6/2024 by Nathan
//  Last tested:  2/1/2024 by Nathan, working as expected.

FUNCTION_BLOCK create_warning
VAR_INPUT
	warning_message: warning_message;
	OK: BOOL;						//  If true, the system is OK.   Assign any and all conditions that are required for the system to be considered 'healthy'.  If this evalutates as FALSE, a warning message is sent.
	time_delay: INT:= 2;			//  A warning message will not be sent unless the problem persists for this long (in seconds.)
END_VAR
VAR_OUTPUT
	warning_sent: BOOL;				//  TRUE if we are in active warning state (and know it.)
END_VAR
VAR
	tracking_problem: BOOL;			//  TRUE if we've seen the "OK" input turn false.
	problem_detected_time: TIME;	//  The time we first saw the problem
	fix_sent: BOOL;					//  TRUE if we've sent a 'fixed' message at least once since rebooting (and must now be sync'd up with the main Warnings list.)
	fix_warning_message: warning_message;	//  Our internally generated (from the warning_message) 'fixed' notification.
END_VAR


IF NOT OK												//  If all of our input conditions are not returning TRUE, something is potentially wrong.
	AND SystemTime.dtDateTime <> DT#1970-01-1-00:00:00	//  Don't begin the process of sending Warnings until our system date/time clock is running.
	AND NOT tracking_problem THEN						//  This statement should only trigger if we aren't already tracking a potential problem (this acts as a rising trigger, creating a timestamp.)
		tracking_problem := TRUE;						//  Note that we are now tracking a problem
		problem_detected_time := TIME();				//  Note the time we first saw the problem.
END_IF

IF OK THEN									//  If the system doesn't see anything wrong,
	tracking_problem := FALSE;				//  note that we aren't actively tracking a problem (any more.)
END_IF

IF tracking_problem													//  If we see a problem
	AND NOT warning_sent											//  and we haven't already sent a warning for this issue
	AND problem_detected_time + time_delay * T#1S < TIME() THEN		//  and it has persisted for at least our specified number of seconds, then
		warnings (warning_message);									//  send our Warning message
		warning_sent := TRUE;										//  Note that we've sent a Warning message
END_IF

IF (warning_sent																			//  If we've previously sent a Warning
	OR NOT fix_sent)																		//  or we may have rebooted and lost track
	AND OK 																					//  and the system now seems to be OK, then: 
	AND SystemTime.dtDateTime <> DT#1970-01-1-00:00:00 THEN									//  Don't begin the process of sending Warnings until our system date/time clock is running.
		fix_warning_message.detail_warning_visu := warning_message.detail_warning_visu;		//  Copy the associated warning visualization name from the main warning message, since that's how the system matches them up.
		fix_warning_message.fixed := TRUE;													//  Set our 'fixed' flag to true, making it a 'fixed' message
		warnings(fix_warning_message);														//  Send our 'fixed' message.  If there isn't a pre-existing matching warning it just gets ignored.
		warning_sent := FALSE;																//  Note that we are no longer in an active warning state
		fix_sent := TRUE;																	//  Note that we have sent a fixed message at least once since rebooting and are now sync'd up with the Warning list.
END_IF

IF warnings_globals.warningSecondaryReset THEN    	//  If the Warning system is signalling that we want to reset all warnings, then:
	tracking_problem:= FALSE;      					//  Reset our 'problem detected' flag
	warning_sent := FALSE;							//  Reset our 'warning sent' flag
	problem_detected_time:= TIME();					//  Reset the time we last saw this issue so it can't instantly trigger when the reset ends.
END_IF

END_FUNCTION_BLOCK

// CR1082/Application/SystemTime
PROGRAM SystemTime
VAR
	getTime: RTCLK.GetDateAndTime;
	setTime: RTCLK.SetDateAndTime;
	dtDateTime: DATE_AND_TIME;
	dwDateTime: DWORD;
	xInit: BOOL;
	tmrGetTime: Ton;
	xGetTime: BOOL;
	dtDate : DATE;
	oldDate : DATE;
	xNewDay : BOOL;
	xLeadLag: BOOL; 
END_VAR
VAR_INPUT
	uiDateTime: DATE_AND_TIME;
	uiDateTime_dw: DWORD;
	xSetTime: BOOL;
END_VAR

tmrGetTime(IN := NOT(tmrGetTime.Q), PT := T#100MS);
//execute gettime every second
xGetTime S= xInit OR tmrGetTime.Q;
getTime(
	xExecute:= xGetTime, 
	xDone=>, 
	xBusy=>, 
	xError=>, 
	eError=>, 
	dtDateAndTime=>, 
	eTimezone=> );
IF xSetTime=0 THEN
	uiDateTime_dw:= TO_DWORD(dtDateTime);
END_IF //changes the user input date time to current time if there is no input
IF getTime.xDone THEN
	xGetTime   := FALSE;
	dtDateTime := getTime.dtDateAndTime;
	dwDateTime := TO_DWORD(getTime.dtDateAndTime);
	
	
END_IF
setTime(
	xExecute:= xSetTime,
	xDone=>,
	xBusy=>,
	xError=>, 
	eError=>,
	dtDateAndTime=> );
uiDateTime:= TO_DT(uiDateTime_dw);
setTime.dtDateAndTime:= uiDateTime;
SystemTime.xSetTime R= setTime.xDone;

dtDate 	:= TO_DATE(dtDateTime);

IF dtDate <> OldDate THEN xNewDay := TRUE;
	ELSE xNewDay := FALSE;
END_IF

xLeadLag S= xNewDay AND NOT(xLeadLag);
xLeadLag R= xNewDay AND		xLeadLag;



oldDate := dtDate;

END_PROGRAM

// CR1082/Application/Pressure_Feed/pressure_transducer_1
//   This program is designed to support a variety of IO-Link pressure transducers.
//   Currently supported:
//		-IFM PM1707 pressure transducer.    https://www.ifm.com/us/en/product/PM1707    Add more sensors if you like.  :-)
//		-IFM PM1789 pressure transducer. 
//		-IFM PV7600 pressure transducer. 
//		-IFM PV7601 pressure transducer. 
//		-IFM PV7602 pressure transducer. 
//		-IFM PV7603 pressure transducer. 	
//		-IFM PV7604 pressure transducer. 


PROGRAM pressure_transducer_1
VAR
	startup_loop_ran: BOOL;		//  We have completed our startup check for the type of level sensor.

	//   WARNINGS
	
	//  Unknown sensor Warning
	
	unknown_sensor_message: warning_message := (red := TRUE, pop_up_everywhere := TRUE, detail_warning_visu := 'W79', short_Description := 'Unknown pressure transducer');
	unknown_sensor_warning: create_warning;

	//  Disconnected sensor Warning

	disconnected_sensor_message: warning_message := (red := TRUE, pop_up_everywhere := TRUE, detail_warning_visu := 'W77', short_Description := 'Pressure transducer disconnected');
	disconnected_sensor_warning: create_warning;

	//  Shorted sensor Warning
		
	shorted_sensor_message: warning_message := (red := TRUE, pop_up_everywhere := TRUE, detail_warning_visu := 'W78', short_Description := 'Pressure transducer shorted');
	shorted_sensor_warning: create_warning;


END_VAR

VAR_INPUT
END_VAR

VAR_OUTPUT
	pressure_psi: REAL;				//  The current pressure in pounds per square inch
	water_depth_inches: REAL;		//  The depth of water needed to produce this pressure
	temperature_F: real;			//  Temp in degrees F, not available for most sensors.
END_VAR

VAR_IN_OUT
	IO_Link_port: IO_link_port;				// Connect to an IO_link read port.   Used to communicate with an analog level sensor, if so equipped.
END_VAR

IF NOT startup_loop_ran THEN pressure_transducer_1.startup_loop(); END_IF			//  This startup loop looks for and identifies what kind of sensor we have available.

analog_warnings_action();   			//  Check all the Warnings associated with these pressure sensors


//   Interpret our data according to the type of sensor:

CASE IO_Link_port.device_ID OF
//	668:  pressure_psi := IO_Link_port.read_word_0 * 0.0014504;			//  PM1707.  Native reading is in tenths of a millibar, this converts to psi.

//	851:  pressure_psi := IO_Link_port.read_word_0 * 1.4504 ;			//  PV7600.  Native reading is in tenths of a bar, this converts to psi.

//	852:  pressure_psi := IO_Link_port.read_word_0 * 1.4504;			//  PV7601.  Native reading is in tenths of a bar, this converts to psi.
	
//	853:  pressure_psi := IO_Link_port.read_word_0 * 0.14504 ;			//  PV7602.  Native reading is in hundredths of a bar, this converts to psi.
	
854:  pressure_psi := IO_Link_port.read_word_0 * 0.14504;			//  PV7603.  Native reading is in hundredths of a bar, this converts to psi.
	
//	855:  pressure_psi := IO_Link_port.read_word_0 * 0.014504;			//  PV7604.  Native reading is in thousandths of a bar, this converts to psi.
	
//   1436:  pressure_psi := IO_Link_port.read_word_0 * 0.00145;			//  PL1506.  Native reading is in tenths of a millibar, this converts to psi.
		  temperature_F := IO_Link_port.read_word_2 * 0.018 + 32;		//  Native reading is in hundredths of a degree C, this converts to F.
		  
		
		  
	  
		//  New sensors can be added here.  Warning code must be updated if you add (for the 'unknown sensor' Warning)
END_CASE

ACTION analog_warnings_action:

//  UNKNOWN SENSOR WARNING!!      This warning checks if the device ID is an unfamiliar one.

	unknown_sensor_warning (OK :=
		IO_Link_port.master_disconnected					//  Don't throw a fault if the master block itself is disconnected
		OR IO_Link_port.not_connected						//  or if nothing is connected to the port (that's a different fault)
		OR (IO_Link_port.vendor_ID = 310
		AND (IO_Link_port.device_ID = 668					//  and we're OK if it's the IFM pressure sensor (PM1707) or
		OR IO_Link_port.device_ID = 670						//  IFM PM1789
		OR IO_Link_port.device_ID = 851						//  IFM PV7600
		OR IO_Link_port.device_ID = 852						//  IFM PV7601
		OR IO_Link_port.device_ID = 853						//  IFM PV7602
		OR IO_Link_port.device_ID = 854						//  IFM PV7603
		OR IO_Link_port.device_ID = 855						//  IFM PV7604
		OR IO_Link_port.device_ID = 1436)),					//  IFM PL1506
		warning_message := unknown_sensor_message,
		time_delay := 15);


//  DEVICE DISCONNECTED WARNING!!  This section checks if no sensor or device is connected.

	disconnected_sensor_warning (OK:=
		IO_Link_port.master_disconnected				//  Don't fault if the master block itself is disconected (so we don't spam the operator with secondary faults when the master is the real problem.)
		OR NOT IO_Link_port.not_connected,				//  We're OK if there hasn't been a 'disconnected' flag set by the master
		warning_message := disconnected_sensor_message,
		time_delay := 10);

//  DEVICE SHORT CIRCUIT WARNING!!	This section checks if a sensor or device is shorted (drawing too much power).

	shorted_sensor_warning (OK :=
		NOT IO_Link_port.short_circuit,					//  We're OK if the master block hasn't reported a short on this port
		warning_message:= shorted_sensor_message);
END_ACTION

END_PROGRAM

// ecomatDisplay43inch_64bit/Application/Pressure_Feed/pressure_transducer_1
//   This program is designed to support a variety of IO-Link pressure transducers.
//   Currently supported:
//		-IFM PM1707 pressure transducer.    https://www.ifm.com/us/en/product/PM1707    Add more sensors if you like.  :-)
//		-IFM PM1789 pressure transducer. 
//		-IFM PV7600 pressure transducer. 
//		-IFM PV7601 pressure transducer. 
//		-IFM PV7602 pressure transducer. 
//		-IFM PV7603 pressure transducer. 	
//		-IFM PV7604 pressure transducer. 


PROGRAM pressure_transducer_1
VAR
	startup_loop_ran: BOOL;		//  We have completed our startup check for the type of level sensor.

	//   WARNINGS
	
	//  Unknown sensor Warning
	
	unknown_sensor_message: warning_message := (red := TRUE, pop_up_everywhere := TRUE, detail_warning_visu := 'W79', short_Description := 'Unknown pressure transducer');
	unknown_sensor_warning: create_warning;

	//  Disconnected sensor Warning

	disconnected_sensor_message: warning_message := (red := TRUE, pop_up_everywhere := TRUE, detail_warning_visu := 'W77', short_Description := 'Pressure transducer disconnected');
	disconnected_sensor_warning: create_warning;

	//  Shorted sensor Warning
		
	shorted_sensor_message: warning_message := (red := TRUE, pop_up_everywhere := TRUE, detail_warning_visu := 'W78', short_Description := 'Pressure transducer shorted');
	shorted_sensor_warning: create_warning;


END_VAR

VAR_INPUT
END_VAR

VAR_OUTPUT
	pressure_psi: REAL;				//  The current pressure in pounds per square inch
	water_depth_inches: REAL;		//  The depth of water needed to produce this pressure
	temperature_F: real;			//  Temp in degrees F, not available for most sensors.
END_VAR

VAR_IN_OUT
	IO_Link_port: IO_link_port;				// Connect to an IO_link read port.   Used to communicate with an analog level sensor, if so equipped.
END_VAR

IF NOT startup_loop_ran THEN pressure_transducer_1.startup_loop(); END_IF			//  This startup loop looks for and identifies what kind of sensor we have available.

analog_warnings_action();   			//  Check all the Warnings associated with these pressure sensors


//   Interpret our data according to the type of sensor:

CASE IO_Link_port.device_ID OF
//	668:  pressure_psi := IO_Link_port.read_word_0 * 0.0014504;			//  PM1707.  Native reading is in tenths of a millibar, this converts to psi.

//	851:  pressure_psi := IO_Link_port.read_word_0 * 1.4504 ;			//  PV7600.  Native reading is in tenths of a bar, this converts to psi.

//	852:  pressure_psi := IO_Link_port.read_word_0 * 1.4504;			//  PV7601.  Native reading is in tenths of a bar, this converts to psi.
	
//	853:  pressure_psi := IO_Link_port.read_word_0 * 0.14504 ;			//  PV7602.  Native reading is in hundredths of a bar, this converts to psi.
	
854:  pressure_psi := IO_Link_port.read_word_0 * 0.14504;			//  PV7603.  Native reading is in hundredths of a bar, this converts to psi.
	
//	855:  pressure_psi := IO_Link_port.read_word_0 * 0.014504;			//  PV7604.  Native reading is in thousandths of a bar, this converts to psi.
	
//   1436:  pressure_psi := IO_Link_port.read_word_0 * 0.00145;			//  PL1506.  Native reading is in tenths of a millibar, this converts to psi.
		  temperature_F := IO_Link_port.read_word_2 * 0.018 + 32;		//  Native reading is in hundredths of a degree C, this converts to F.
		  
		
		  
	  
		//  New sensors can be added here.  Warning code must be updated if you add (for the 'unknown sensor' Warning)
END_CASE

END_PROGRAM

// CR1082/Application/IO Blocks/AL1342 Master block/AL1342_IO_Link_Master_A
//  This program creates an abstraction layer for an AL1342 IO-Link master block (or similar.)   This layer allows software to be easily reconfigured in
//  CFC and other 'top level' programs by simply switching a couple input/output variables.


PROGRAM AL1342_IO_Link_Master_A
VAR
	startup_ran: BOOL;


	//   WARNINGS
	
	//   Disconnected master block Warning

	disconnected_master_message: warning_message := (red := TRUE, pop_up_everywhere := TRUE, detail_warning_visu := 'W30', short_Description := 'Master block disconnected');
	
	disconnected_master_warning: create_warning;
		

		
END_VAR

VAR_OUTPUT
	X_null: IO_link_port;	//  A 'dead' port; reading and writing to it has no effect.  This is used for objects that have an in/out IO-Link port (so they need something connected to avoid angering the compiler) but aren't using that port for the current application.
	X_01: IO_link_port;		//  Data from port X-01 on block AL1342 (first or only Master.)
	X_02: IO_link_port;		//  Data from port X-02 on block AL1342 (first or only Master.)
	X_03: IO_link_port;		//  Data from port X-03 on block AL1342 (first or only Master.)
	X_04: IO_link_port;		//  Data from port X-04 on block AL1342 (first or only Master.)
	X_05: IO_link_port;		//  Data from port X-05 on block AL1342 (first or only Master.)
	X_06: IO_link_port;		//  Data from port X-06 on block AL1342 (first or only Master.)
	X_07: IO_link_port;		//  Data from port X-07 on block AL1342 (first or only Master.)
	X_08: IO_link_port;		//  Data from port X-08 on block AL1342 (first or only Master.)	
END_VAR

VAR_IN_OUT
	
END_VAR


//  Startup by populating some information that only gets set once.

IF NOT startup_ran THEN
	X_01.block_name := 'AL1342';
	X_02.block_name := 'AL1342';
	X_03.block_name := 'AL1342';
	X_04.block_name := 'AL1342';
	X_05.block_name := 'AL1342';
	X_06.block_name := 'AL1342';
	X_07.block_name := 'AL1342';
	X_08.block_name := 'AL1342';

	X_01.port_ID := 'X01';
	X_02.port_ID := 'X02';
	X_03.port_ID := 'X03';
	X_04.port_ID := 'X04';
	X_05.port_ID := 'X05';
	X_06.port_ID := 'X06';
	X_07.port_ID := 'X07';
	X_08.port_ID := 'X08';
	
	X_01.port_number := 1;
	X_02.port_number := 2;
	X_03.port_number := 3;
	X_04.port_number := 4;
	X_05.port_number := 5;
	X_06.port_number := 6;
	X_07.port_number := 7;
	X_08.port_number := 8;
	
	startup_ran := TRUE;
END_IF


//    Populate the data fields of the various input/output structs.

//  Read vendor/device IDs:

	X_01.vendor_ID := AL1342_X01_vendorID;
	X_02.vendor_ID := AL1342_X02_vendorID;
	X_03.vendor_ID := AL1342_X03_vendorID;
	X_04.vendor_ID := AL1342_X04_vendorID;
	X_05.vendor_ID := AL1342_X05_vendorID;
	X_06.vendor_ID := AL1342_X06_vendorID;
	X_07.vendor_ID := AL1342_X07_vendorID;
	X_08.vendor_ID := AL1342_X08_vendorID;
	
	X_01.device_ID := AL1342_X01_deviceID;
	X_02.device_ID := AL1342_X02_deviceID;
	X_03.device_ID := AL1342_X03_deviceID;
	X_04.device_ID := AL1342_X04_deviceID;
	X_05.device_ID := AL1342_X05_deviceID;
	X_06.device_ID := AL1342_X06_deviceID;
	X_07.device_ID := AL1342_X07_deviceID;
	X_08.device_ID := AL1342_X08_deviceID;

//  Read in digital input pins.  These inputs only function if the port is configured as an input.

	X_01.DI_pin_4 := AL1342_read_X01_DI_pin4;
	X_01.DI_pin_2 := AL1342_read_X01_DI_pin2;

	X_02.DI_pin_4 := AL1342_read_X02_DI_pin4;
	X_02.DI_pin_2 := AL1342_read_X02_DI_pin2;
	
	X_03.DI_pin_4 := AL1342_read_X03_DI_pin4;
	X_03.DI_pin_2 := AL1342_read_X03_DI_pin2;
	
	X_04.DI_pin_4 := AL1342_read_X04_DI_pin4;
	X_04.DI_pin_2 := AL1342_read_X04_DI_pin2;
	
	X_05.DI_pin_4 := AL1342_read_X05_DI_pin4;
	X_05.DI_pin_2 := AL1342_read_X05_DI_pin2;
	
	X_06.DI_pin_4 := AL1342_read_X06_DI_pin4;
	X_06.DI_pin_2 := AL1342_read_X06_DI_pin2;
	
	X_07.DI_pin_4 := AL1342_read_X07_DI_pin4;
	X_07.DI_pin_2 := AL1342_read_X07_DI_pin2;
	
	X_08.DI_pin_4 := AL1342_read_X08_DI_pin4;
	X_08.DI_pin_2 := AL1342_read_X08_DI_pin2;
	
//  Read in short circuit messages

	X_01.short_circuit := X01_shortcircuit;
	X_02.short_circuit := X02_shortcircuit;
	X_03.short_circuit := X03_shortcircuit;
	X_04.short_circuit := X04_shortcircuit;
	X_05.short_circuit := X05_shortcircuit;
	X_06.short_circuit := X06_shortcircuit;
	X_07.short_circuit := X07_shortcircuit;
	X_08.short_circuit := X08_shortcircuit;

//  Read in status messages (port disconnected or data corrupt)

	X_01.not_connected := AL1342_X01_not_connected;
	X_01.data_invalid := X01_data_invalid;
	
	X_02.not_connected := AL1342_X02_not_connected;
	X_02.data_invalid := X02_data_invalid;
	
	X_03.not_connected := AL1342_X03_not_connected;
	X_03.data_invalid := X03_data_invalid;
	
	X_04.not_connected := AL1342_X04_not_connected;
	X_04.data_invalid := X04_data_invalid;
	
	X_05.not_connected := X05_not_connected;
	X_05.data_invalid := X05_data_invalid;

	X_06.not_connected := X06_not_connected;
	X_06.data_invalid := X06_data_invalid;
	
	X_07.not_connected := X07_not_connected;
	X_07.data_invalid := X07_data_invalid;
	
	X_08.not_connected := X08_not_connected;
	X_08.data_invalid := X08_data_invalid;
	
	
//  Read IO-Link process data words

	X_01.read_word_0 := AL1342_read_X01_word_0;
	X_01.read_word_1 := AL1342_read_X01_word_1;
	X_01.read_word_2 := AL1342_read_X01_word_2;
	X_01.read_word_3 := AL1342_read_X01_word_3;
	X_01.read_word_4 := AL1342_read_X01_word_4;
	X_01.read_word_5 := AL1342_read_X01_word_5;
	X_01.read_word_6 := AL1342_read_X01_word_6;

	X_02.read_word_0 := AL1342_read_X02_word_0;
	X_02.read_word_1 := AL1342_read_X02_word_1;
	X_02.read_word_2 := AL1342_read_X02_word_2;
	X_02.read_word_3 := AL1342_read_X02_word_3;
	X_02.read_word_4 := AL1342_read_X02_word_4;
	X_02.read_word_5 := AL1342_read_X02_word_5;
	X_02.read_word_6 := AL1342_read_X02_word_6;

	X_03.read_word_0 := AL1342_read_X03_word_0;
	X_03.read_word_1 := AL1342_read_X03_word_1;
	X_03.read_word_2 := AL1342_read_X03_word_2;
	X_03.read_word_3 := AL1342_read_X03_word_3;
	X_03.read_word_4 := AL1342_read_X03_word_4;
	X_03.read_word_5 := AL1342_read_X03_word_5;
	X_03.read_word_6 := AL1342_read_X03_word_6;
	
	X_04.read_word_0 := AL1342_read_X04_word_0;
	X_04.read_word_1 := AL1342_read_X04_word_1;
	X_04.read_word_2 := AL1342_read_X04_word_2;
	X_04.read_word_3 := AL1342_read_X04_word_3;
	X_04.read_word_4 := AL1342_read_X04_word_4;
	X_04.read_word_5 := AL1342_read_X04_word_5;
	X_04.read_word_6 := AL1342_read_X04_word_6;
	
	X_05.read_word_0 := AL1342_read_X05_word_0;
	X_05.read_word_1 := AL1342_read_X05_word_1;
	X_05.read_word_2 := AL1342_read_X05_word_2;
	X_05.read_word_3 := AL1342_read_X05_word_3;
	X_05.read_word_4 := AL1342_read_X05_word_4;
	X_05.read_word_5 := AL1342_read_X05_word_5;
	X_05.read_word_6 := AL1342_read_X05_word_6;
	
	X_06.read_word_0 := AL1342_read_X06_word_0;
	X_06.read_word_1 := AL1342_read_X06_word_1;
	X_06.read_word_2 := AL1342_read_X06_word_2;
	X_06.read_word_3 := AL1342_read_X06_word_3;
	X_06.read_word_4 := AL1342_read_X06_word_4;
	X_06.read_word_5 := AL1342_read_X06_word_5;
	X_06.read_word_6 := AL1342_read_X06_word_6;
	
	X_07.read_word_0 := AL1342_read_X07_word_0;
	X_07.read_word_1 := AL1342_read_X07_word_1;
	X_07.read_word_2 := AL1342_read_X07_word_2;
	X_07.read_word_3 := AL1342_read_X07_word_3;
	X_07.read_word_4 := AL1342_read_X07_word_4;
	X_07.read_word_5 := AL1342_read_X07_word_5;
	X_07.read_word_6 := AL1342_read_X07_word_6;

	X_08.read_word_0 := AL1342_read_X08_word_0;
	X_08.read_word_1 := AL1342_read_X08_word_1;
	X_08.read_word_2 := AL1342_read_X08_word_2;
	X_08.read_word_3 := AL1342_read_X08_word_3;
	X_08.read_word_4 := AL1342_read_X08_word_4;
	X_08.read_word_5 := AL1342_read_X08_word_5;
	X_08.read_word_6 := AL1342_read_X08_word_6;


//   WRITE data out to the IO-Link port
	
	AL1342_write_X01_word_0 := X_01.write_word_0;
	AL1342_write_X01_word_1 := X_01.write_word_1;
	AL1342_write_X01_word_2 := X_01.write_word_2;
	AL1342_write_X01_word_3 := X_01.write_word_3;

	AL1342_write_X02_word_0 := X_02.write_word_0;
	AL1342_write_X02_word_1 := X_02.write_word_1;
	AL1342_write_X02_word_2 := X_02.write_word_2;
	AL1342_write_X02_word_3 := X_02.write_word_3;
	
	AL1342_write_X03_word_0 := X_03.write_word_0;
	AL1342_write_X03_word_1 := X_03.write_word_1;
	AL1342_write_X03_word_2 := X_03.write_word_2;
	AL1342_write_X03_word_3 := X_03.write_word_3;
	
	AL1342_write_X04_word_0 := X_04.write_word_0;
	AL1342_write_X04_word_1 := X_04.write_word_1;
	AL1342_write_X04_word_2 := X_04.write_word_2;
	AL1342_write_X04_word_3 := X_04.write_word_3;
	
	AL1342_write_X05_word_0 := X_05.write_word_0;
	AL1342_write_X05_word_1 := X_05.write_word_1;
	AL1342_write_X05_word_2 := X_05.write_word_2;
	AL1342_write_X05_word_3 := X_05.write_word_3;
	
	AL1342_write_X06_word_0 := X_06.write_word_0;
	AL1342_write_X06_word_1 := X_06.write_word_1;
	AL1342_write_X06_word_2 := X_06.write_word_2;
	AL1342_write_X06_word_3 := X_06.write_word_3;
	
	AL1342_write_X07_word_0 := X_07.write_word_0;
	AL1342_write_X07_word_1 := X_07.write_word_1;
	AL1342_write_X07_word_2 := X_07.write_word_2;
	AL1342_write_X07_word_3 := X_07.write_word_3;
	
	AL1342_write_X08_word_0 := X_08.write_word_0;
	AL1342_write_X08_word_1 := X_08.write_word_1;
	AL1342_write_X08_word_2 := X_08.write_word_2;
	AL1342_write_X08_word_3 := X_08.write_word_3;
	
	
	//  Write digital outputs (1 DO per port, only available if the port is configured as an output.)
	
	AL1342_write_X01_pin4 := X_01.DO_pin_4;
	AL1342_write_X02_pin4 := X_02.DO_pin_4;
	AL1342_write_X03_pin4 := X_03.DO_pin_4;
	AL1342_write_X04_pin4 := X_04.DO_pin_4;
	AL1342_write_X05_pin4 := X_05.DO_pin_4;
	AL1342_write_X06_pin4 := X_06.DO_pin_4;
	AL1342_write_X07_pin4 := X_07.DO_pin_4;
	AL1342_write_X08_pin4 := X_08.DO_pin_4;
	
	//  Set master block disconnect status
	
	X_01.master_disconnected := AL1342.ComState <> 2;
	X_02.master_disconnected := AL1342.ComState <> 2;
	X_03.master_disconnected := AL1342.ComState <> 2;
	X_04.master_disconnected := AL1342.ComState <> 2;
	X_05.master_disconnected := AL1342.ComState <> 2;
	X_06.master_disconnected := AL1342.ComState <> 2;
	X_07.master_disconnected := AL1342.ComState <> 2;
	X_08.master_disconnected := AL1342.ComState <> 2;
	
	
//    WARNINGS       WARNINGS     WARNINGS

//  Master block disconnected warning

disconnected_master_warning (OK :=
	AL1342.ComState = 2,								//  Connection state 2 is connected and communicating normally, so if we see that, we're good.
	warning_message := disconnected_master_message);

END_PROGRAM

// CR1082/Application/Sentronic/Feed_Diaphram_Pump
PROGRAM Feed_Diaphram_Pump
VAR
	hand_run_mixer: BOOL;					//  True if somebody is pressing the button to hand run the mixer.
		//   WARNINGS
	
	//  VFD not responding Warning.

	mixer_VFD_not_responding_message: warning_message := (red := TRUE, pop_up_everywhere := TRUE, detail_warning_visu := 'W???', short_Description := 'Pit mixer VFD not responding');
	
	mixer_VFD_not_responding_warning: create_warning;

	//  Unknown device Warning
	
	unknown_device_message: warning_message := (red := TRUE, pop_up_everywhere := TRUE, detail_warning_visu := 'W???', short_Description := 'Unknown pit mixer adapter');
	
	unknown_device_warning: create_warning;
	
	//   Disconnected device Warning

	disconnected_adapter_message: warning_message := (red := TRUE, pop_up_everywhere := TRUE, detail_warning_visu := 'W???',short_Description := 'Pit mixer adapter disconnected');
	
	disconnected_adapter_warning: create_warning;
	
	//  Shorted device Warning

	shorted_device_message: warning_message := (red := TRUE, pop_up_everywhere := TRUE, detail_warning_visu := 'W???', short_Description := 'Pit mixer adapter shorted');
	
	shorted_device_warning: create_warning;


END_VAR
VAR_INPUT
Sentronic_Real: REAL;
END_VAR
	

VAR_IN_OUT
	DP1213_IO_link: IO_link_port;
END_VAR


//  Turn our VFD enable output on or off depending on whether or not there's a request for the mixer to run:



//  Convert our 0-100% to a 4-20 mA signal and send it to the correct word of the IO-link D/A converter

// 

DP1213_IO_link.write_word_0 := TO_WORD(Sentronic_Real);
DP1213_IO_link.write_word_1 := TO_WORD(Sentronic_Real);

//    WARNINGS       WARNINGS     WARNINGS

//   VFD not responding warning

mixer_VFD_not_responding_warning (OK :=,
//	NOT VFD_enable											//   We are OK if we either aren't trying to run the VFD,
//	OR VFD_feedback,										//   or if we see a signal that the VFD is running.
	warning_message := mixer_VFD_not_responding_message,
	time_delay:= 5);


//  UNKNOWN DEVICE WARNING!!      This warning checks if the device ID of our digital to analog adapter (used to send the 4-20 mA speed signal) is an unfamiliar one.

unknown_device_warning (OK:=
	DP1213_IO_link.not_connected				//  Don't fault if nothing at all is connected (that's a different warning.)
	OR DP1213_IO_link.master_disconnected		//  Don't fault if the master is disconnected (to avoid spamming the operator with secondary disconnects when the master disconnect is the real problem.)
	OR (DP1213_IO_link.device_ID = 612			//  and of course we are OK if we do see the expected IFM DP1213 adapter.
	AND DP1213_IO_link.vendor_ID = 310),
	warning_message:= unknown_device_message,
	time_delay := 10);
	

//  DEVICE DISCONNECTED WARNING!!   This section checks if our DP1312 (D/A converter) is connected.

disconnected_adapter_warning (OK:=
	NOT DP1213_IO_link.not_connected			//  We are OK if the master block isn't reporting a disconnect or communication problem.
	AND NOT DP1213_IO_link.data_invalid,
	warning_message:= disconnected_adapter_message,
	time_delay := 10);


//  DEVICE SHORT CIRCUIT WARNING!!

shorted_device_warning (OK :=
	NOT DP1213_IO_link.short_circuit,
	warning_message := shorted_device_message);

END_PROGRAM

// ecomatDisplay43inch_64bit/Application/Sentronic/Feed_Diaphram_Pump
PROGRAM Feed_Diaphram_Pump
VAR
	hand_run_mixer: BOOL;					//  True if somebody is pressing the button to hand run the mixer.
		//   WARNINGS
	
	//  VFD not responding Warning.

	mixer_VFD_not_responding_message: warning_message := (red := TRUE, pop_up_everywhere := TRUE, detail_warning_visu := 'W???', short_Description := 'Pit mixer VFD not responding');
	
	mixer_VFD_not_responding_warning: create_warning;

	//  Unknown device Warning
	
	unknown_device_message: warning_message := (red := TRUE, pop_up_everywhere := TRUE, detail_warning_visu := 'W???', short_Description := 'Unknown pit mixer adapter');
	
	unknown_device_warning: create_warning;
	
	//   Disconnected device Warning

	disconnected_adapter_message: warning_message := (red := TRUE, pop_up_everywhere := TRUE, detail_warning_visu := 'W???',short_Description := 'Pit mixer adapter disconnected');
	
	disconnected_adapter_warning: create_warning;
	
	//  Shorted device Warning

	shorted_device_message: warning_message := (red := TRUE, pop_up_everywhere := TRUE, detail_warning_visu := 'W???', short_Description := 'Pit mixer adapter shorted');
	
	shorted_device_warning: create_warning;


END_VAR
VAR_INPUT
Sentronic_Real: REAL;
END_VAR
	

VAR_IN_OUT
	DP1213_IO_link: IO_link_port;
END_VAR


//  Turn our VFD enable output on or off depending on whether or not there's a request for the mixer to run:



//  Convert our 0-100% to a 4-20 mA signal and send it to the correct word of the IO-link D/A converter

// 

DP1213_IO_link.write_word_0 := TO_WORD(Sentronic_Real);
DP1213_IO_link.write_word_1 := TO_WORD(Sentronic_Real);

//    WARNINGS       WARNINGS     WARNINGS

//   VFD not responding warning

mixer_VFD_not_responding_warning (OK :=,
//	NOT VFD_enable											//   We are OK if we either aren't trying to run the VFD,
//	OR VFD_feedback,										//   or if we see a signal that the VFD is running.
	warning_message := mixer_VFD_not_responding_message,
	time_delay:= 5);


//  UNKNOWN DEVICE WARNING!!      This warning checks if the device ID of our digital to analog adapter (used to send the 4-20 mA speed signal) is an unfamiliar one.

unknown_device_warning (OK:=
	DP1213_IO_link.not_connected				//  Don't fault if nothing at all is connected (that's a different warning.)
	OR DP1213_IO_link.master_disconnected		//  Don't fault if the master is disconnected (to avoid spamming the operator with secondary disconnects when the master disconnect is the real problem.)
	OR (DP1213_IO_link.device_ID = 612			//  and of course we are OK if we do see the expected IFM DP1213 adapter.
	AND DP1213_IO_link.vendor_ID = 310),
	warning_message:= unknown_device_message,
	time_delay := 10);
	

//  DEVICE DISCONNECTED WARNING!!   This section checks if our DP1312 (D/A converter) is connected.

disconnected_adapter_warning (OK:=
	NOT DP1213_IO_link.not_connected			//  We are OK if the master block isn't reporting a disconnect or communication problem.
	AND NOT DP1213_IO_link.data_invalid,
	warning_message:= disconnected_adapter_message,
	time_delay := 10);


//  DEVICE SHORT CIRCUIT WARNING!!

shorted_device_warning (OK :=
	NOT DP1213_IO_link.short_circuit,
	warning_message := shorted_device_message);

END_PROGRAM

// CR1082/Application/PROGRAM_ROUTINES/POU_MANUAL_CONTROL
PROGRAM POU_MANUAL_CONTROL
VAR
END_VAR

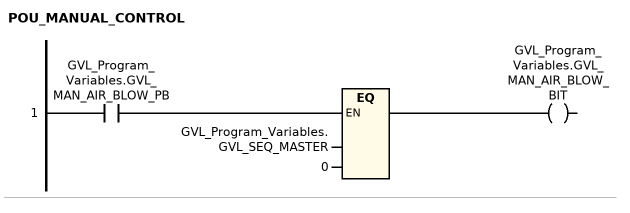
// NETWORK 1
GVL_Program_Variables.GVL_MAN_AIR_BLOW_BIT := GVL_Program_Variables.GVL_MAN_AIR_BLOW_PB AND GVL_Program_Variables.GVL_SEQ_MASTER = 0;

END_PROGRAM

// CR1082/Application/Sentronic/POU_Sentronic_ST
PROGRAM POU_Sentronic_ST
VAR
END_VAR

AL1342_IO_Link_Master_A.X_08.write_word_0 := TO_WORD(pvars.Sentronic_Real);

END_PROGRAM

// ecomatDisplay43inch_64bit/Application/Sentronic/POU_Sentronic_ST
PROGRAM POU_Sentronic_ST
VAR
END_VAR

AL1342_IO_Link_Master_A.X_08.write_word_0 := TO_WORD(pvars.Sentronic_Real);

END_PROGRAM

// CR1082/Application/Warning system/visu_context
PROGRAM visu_context
VAR
	previousvisu: STRING := 'null';						//   The last visualization we responded to.  Used to prevent the code from triggering when nothing has changed.  Pre-loaded with 'null'
														//   so the system will trigger on initial startup.   (Otherwise the button lights are wrong until after the first visu change.)
	option_clicks: INT;									//   This tracks how many times somebody has pressed the right arrow button while in the Options screen.   Used to decide when to show the hidden config button.
	myCounter: INT;										//   Used for some loops
			//  The function block that adjusts screen brightness.
	startup_ran: BOOL;									//  Turn to TRUE after we complete any startup tasks.
	show_detail_screen: BOOL;

	change_splash_screen: BOOL;							//  Install a new splash screen.
	new_software_version_notice: warning_message := (informational := TRUE, detail_warning_visu := 'W173', short_Description := 'System software updated');
		//  This struct contains the actual color settings and on/off settings for the physical button backlights.
	flasher: BOOL;											//  Turns the warning button lights on and off.
	flash_time: TIME;
END_VAR
VAR_INPUT
	update_now: BOOL:= 1;								//  Set to TRUE to cause the button lights to update without a change in visu.
END_VAR

(* This program handles some interface tasks.  It:

- Changes the button lights (on/off and color) depending on which buttons are active and various status conditions.
- Turns off the audible alarm if you go to the Warnings screen.
- Displays contextual popups if there's an active Warning and the user has navigated to the corresponding screen.
- Generates a notification if the software version has changed.

Each visualization screen gets its own IF/THEN statement and set of button light settings.   Sadly, CASE does not support strings in structured text.
*)
	



IF NOT (pvars.redWarningPresent				//  If we don't have any active warnings, then just leave the warning log button light on.
	OR pvars.yellowWarningPresent
	OR pvars.blueWarningPresent) THEN
		flasher := TRUE;
END_IF


IF VisuElems.CurrentVisu <> previousvisu		//  Has the visualization changed?
	OR update_now THEN							//  Or has a manual update been requested?   If so:
		update_now := FALSE;					//  Reset our manual update trigger and run through the whole context sequence...

	//  If the flag is set for a contextual Warning pop-up, switch to that Warning detail screen, then disable the flag.

	FOR myCounter := 16 TO 1 BY -1 DO
		IF (pVars.myWarnings[myCounter].contextual_visu = VisuElems.CurrentVisu)			//  Is there a warning set to pop-up on the current screen?
			AND (pVars.myWarnings [myCounter].fixed = FALSE)								//  Is it unfixed?  (We don't want to pop-up a warning on things that aren't relevent any more!)
			AND pVars.myWarnings[myCounter].pop_up_contextual = TRUE THEN					//  If this warning is set to create a contextual pop-up
				VisuElems.CurrentVisu := pVars.myWarnings[myCounter].detail_warning_visu;   //  Set the current visualization to the warning detail visualization for that Warning.
				pVars.myWarnings[myCounter].pop_up_contextual := FALSE;						//  Clear our flag to pop up contextually so it doesn't keep happening.
		END_IF
	END_FOR
	
	
	
	
	previousvisu := VisuElems.CurrentVisu;

END_IF

END_PROGRAM

// CR1082/Application/Main/Graph
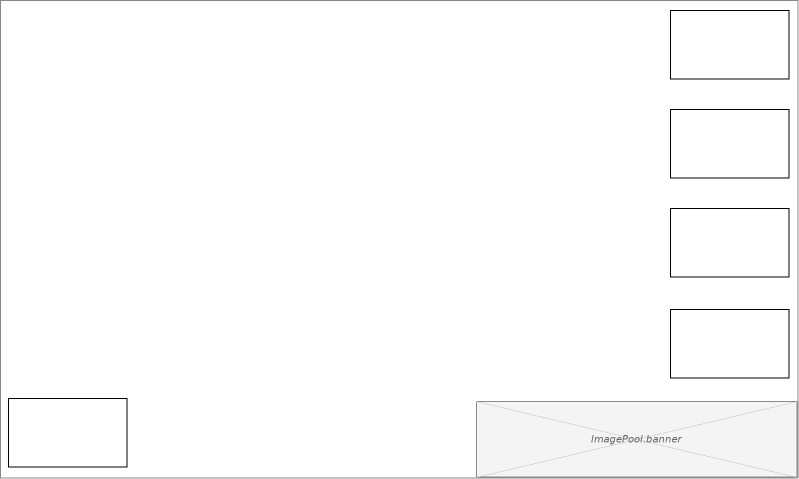
VISUALIZATION Graph  // 799x479, background image ImagePool.background
    Image (476,401 321x76), image: ImagePool.banner
    Label (254,8 266x62), "Graph Screen"
    Rectangle (670,10 119x69), "SETPOINT"
    Rectangle (670,109 119x69), "MANUAL"
    Rectangle (670,208 119x69), "GRAPH"
    Rectangle (670,309 119x69), "STATS"
    Rectangle (8,398 119x69), "MAIN"
    hotkey  Id=481041580032, Key=KeyDown=True, KeyName=KEY3_1, ActionToExecute=Action=Assign=Stats, Type=Assignment, VisuElemId=-1
    hotkey  Id=481040531456, Key=KeyDown=True, KeyName=KEY3_2, ActionToExecute=Action=Assign=Graph, Type=Assignment, VisuElemId=-1
    hotkey  Id=481039482880, Key=KeyDown=True, KeyName=KEY3_3, ActionToExecute=Action=Assign=Manual, Type=Assignment, VisuElemId=-1
    hotkey  Id=481038434304, Key=KeyDown=True, KeyName=KEY3_4, ActionToExecute=Action=Assign=Setpoints, Type=Assignment, VisuElemId=-1
    hotkey  Id=481037385728, Key=KeyDown=True, KeyName=KEY1_5, ActionToExecute=Action=Assign=Main_Screen, Type=Assignment, VisuElemId=-1
END_VISUALIZATION

// CR1082/Application/Main/Main_Screen
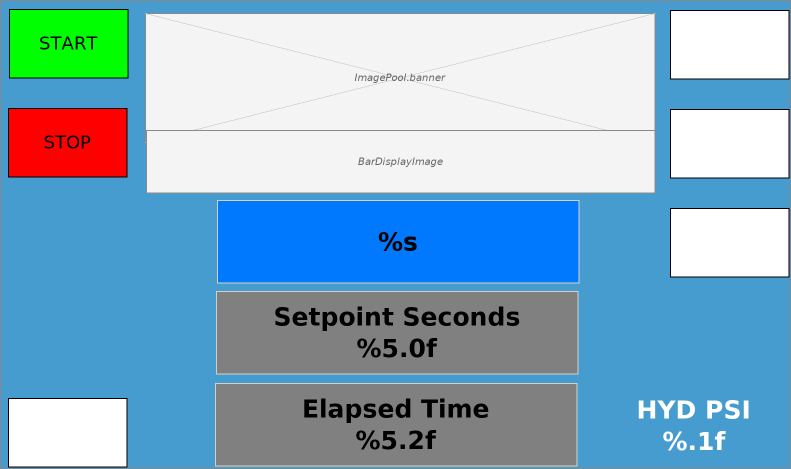
VISUALIZATION Main_Screen  // 791x469, background image ImagePool.background
    Image (145,13 510x129), image: ImagePool.banner
    Rectangle (670,10 119x69), "SETPOINT"
    Rectangle (670,109 119x69), "MANUAL"
    Rectangle (670,208 119x69), "STATS"
    Rectangle (8,398 119x69), "MAIN"
    Rectangle (8,108 119x69), "STOP"
    Rectangle (9,9 119x69), "START"
    BarDisplayImage (146,130 509x63), value: pressure_transducer_1.pressure_psi, style: BarDisplayImage-Gray, scale format: %.1f, scale 0..100
        p518627256: Cake PSI
    Textfield (217,200 362x83), "%s", text variable: POU_aSeq_Master.Message_String
    Textfield (216,291 362x83), "Setpoint Seconds %5.0f", text variable: GVL_Program_Variables.GVL_DISPLAY_SETPOINT
    Textfield (215,383 362x83), "Elapsed Time %5.2f", text variable: GVL_Program_Variables.GVL_DISPLAY_TIME
    Textfield (601,384 186x83), "HYD PSI %.1f", text variable: pressure_transducer.pressure_psi
    hotkey  Id=481040531456, Key=KeyDown=True, KeyName=KEY3_2, ActionToExecute=Action=Assign=Stats, Type=Assignment, VisuElemId=-1
    hotkey  Id=481039482880, Key=KeyDown=True, KeyName=KEY3_3, ActionToExecute=Action=Assign=Manual, Type=Assignment, VisuElemId=-1
    hotkey  Id=481038434304, Key=KeyDown=True, KeyName=KEY3_4, ActionToExecute=Action=Assign=Setpoints, Type=Assignment, VisuElemId=-1
    hotkey  Id=481037385728, Key=KeyDown=True, KeyName=KEY1_5, ActionToExecute=Action=Assign=Main_Screen, Type=Assignment, VisuElemId=-1
    hotkey  Id=481047871488, Key=KeyDown=True, KeyName=KEY1_2, ActionToExecute=Action=STSnippet=GVL_PROGRAM_VARIABLES.GVL_STOP_PB:=TRUE;, VisuElemId=-1
    hotkey  Id=481046822912, Key=KeyName=KEY1_2, ActionToExecute=Action=STSnippet=GVL_PROGRAM_VARIABLES.GVL_STOP_PB:=FALSE;, VisuElemId=-1
    hotkey  Id=481045774336, Key=KeyDown=True, KeyName=KEY1_1, ActionToExecute=Action=STSnippet=GVL_PROGRAM_VARIABLES.GVL_START_PB:=TRUE;, VisuElemId=-1
    hotkey  Id=481044725760, Key=KeyName=KEY1_1, ActionToExecute=Action=STSnippet=GVL_PROGRAM_VARIABLES.GVL_START_PB:=FALSE;, VisuElemId=-1
END_VISUALIZATION

// CR1082/Application/Main/Manual
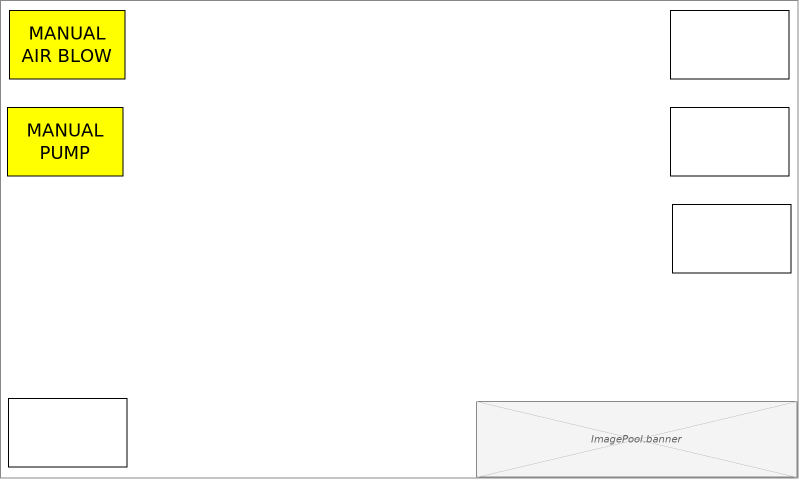
VISUALIZATION Manual  // 799x479, background image ImagePool.background
VAR
	
scale_low: REAL;
scale_high: REAL:= 4500.0;
	
END_VAR
    Rectangle (670,10 119x69), "SETPOINT"
    Rectangle (670,107 119x69), "MANUAL"
    Rectangle (672,204 119x69), "STATS"
    Rectangle (8,398 119x69), "MAIN"
    Image (476,401 321x76), image: ImagePool.banner
    Label (246,14 305x63), "Manual Screen"
    Rectangle (9,10 116x69), "MANUAL AIR BLOW", colour toggle: GVL_Program_Variables.GVL_MAN_AIR_BLOW_PB
    Rectangle (7,107 116x69), "MANUAL PUMP", colour toggle: GVL_Program_Variables.GVL_MAN_DIAPHRAM_PUMP
    hotkey  Id=481040531456, Key=KeyDown=True, KeyName=KEY3_2, ActionToExecute=Action=Assign=Stats, Type=Assignment, VisuElemId=-1
    hotkey  Id=481039482880, Key=KeyDown=True, KeyName=KEY3_3, ActionToExecute=Action=Assign=Manual, Type=Assignment, VisuElemId=-1
    hotkey  Id=481038434304, Key=KeyDown=True, KeyName=KEY3_4, ActionToExecute=Action=Assign=Setpoints, Type=Assignment, VisuElemId=-1
    hotkey  Id=481037385728, Key=KeyDown=True, KeyName=KEY1_5, ActionToExecute=Action=Assign=Main_Screen, Type=Assignment, VisuElemId=-1
    hotkey  Id=481043677184, Key=KeyDown=True, KeyName=KEY1_1, ActionToExecute=Action=STSnippet=GVL_Program_Variables.GVL_MAN_AIR_BLOW_PB := 1;, VisuElemId=-1
    hotkey  Id=481044725760, Key=KeyName=KEY1_1, ActionToExecute=Action=STSnippet=GVL_Program_Variables.GVL_MAN_AIR_BLOW_PB := 0;, VisuElemId=-1
    hotkey  Id=481045774336, Key=KeyDown=True, KeyName=KEY1_2, ActionToExecute=Action=STSnippet=GVL_PROGRAM_VARIABLES.GVL_MAN_DIAPHRAM_PUMP := 1;, VisuElemId=-1
    hotkey  Id=481046822912, Key=KeyName=KEY1_2, ActionToExecute=Action=STSnippet=GVL_PROGRAM_VARIABLES.GVL_MAN_DIAPHRAM_PUMP := 0;, VisuElemId=-1
END_VISUALIZATION

// CR1082/Application/Main/Setpoints
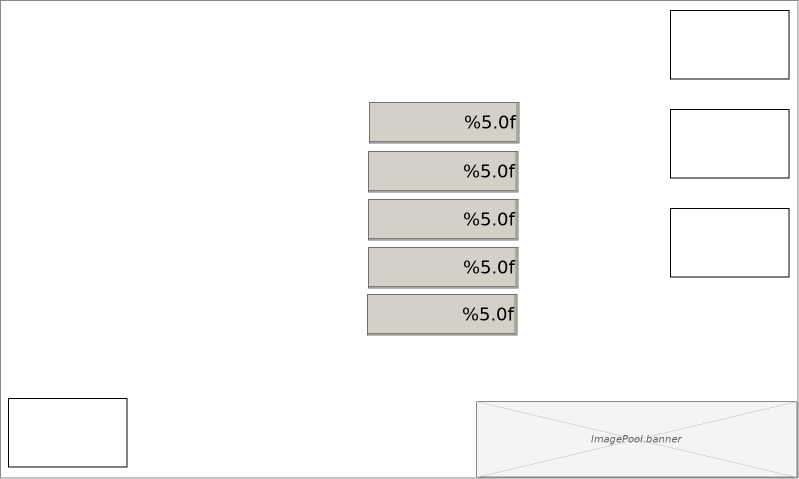
VISUALIZATION Setpoints  // 799x479, background image ImagePool.background
    Rectangle (670,10 119x69), "SETPOINT"
    Rectangle (670,109 119x69), "MANUAL"
    Rectangle (670,208 119x69), "STATS"
    Rectangle (8,398 119x69), "MAIN"
    Image (476,401 321x76), image: ImagePool.banner
    Label (220,9 351x49), "Setpoints Screen"
    Button (369,102 150x41), "%5.0f", text variable: pVars.Hydraulic_PSI_Setpoint
        OnMouseClick: write pVars.Hydraulic_PSI_Setpoint via VisuDialogs.Numpad, min 0, max 4500
    Label (101,102 261x40), "Hyd Close Pressure 0-4500"
    Button (368,151 150x41), "%5.0f", text variable: pVars.Cake_Feed_PSI_Setpoint
        OnMouseClick: write pVars.Cake_Feed_PSI_Setpoint via VisuDialogs.Numpad, min 0, max 100
    Label (100,151 261x40), "Cake Feed Pressure 0-100"
    Button (368,199 150x41), "%5.0f", text variable: pVars.Air_Blow_Minutes
        OnMouseClick: write pVars.Air_Blow_Minutes via VisuDialogs.Numpad, min 0, max 720
    Label (100,199 261x40), "Air Blow Time (Min)"
    Button (368,247 150x41), "%5.0f", text variable: pVars.Cake_Feed_Time_Delay_Secs
        OnMouseClick: write pVars.Cake_Feed_Time_Delay_Secs via VisuDialogs.Numpad, min 0, max 999
    Label (78,247 283x40), "Cake Done Time Delay (Min)"
    Button (367,294 150x41), "%5.0f", text variable: pVars.Cake_Stepup_Factor
        OnMouseClick: write pVars.Cake_Stepup_Factor via VisuDialogs.Numpad, min 0, max 2000
    Label (59,294 301x40), "Cake Stepup Factor 0-2000"
    hotkey  Id=481038434304, Key=KeyDown=True, KeyName=KEY3_2, ActionToExecute=Action=Assign=Stats, Type=Assignment, VisuElemId=-1
    hotkey  Id=481039482880, Key=KeyDown=True, KeyName=KEY3_3, ActionToExecute=Action=Assign=Manual, Type=Assignment, VisuElemId=-1
    hotkey  Id=481040531456, Key=KeyDown=True, KeyName=KEY3_4, ActionToExecute=Action=Assign=Setpoints, Type=Assignment, VisuElemId=-1
    hotkey  Id=481041580032, Key=KeyDown=True, KeyName=KEY1_5, ActionToExecute=Action=Assign=Main_Screen, Type=Assignment, VisuElemId=-1
END_VISUALIZATION

// CR1082/Application/Main/Stats
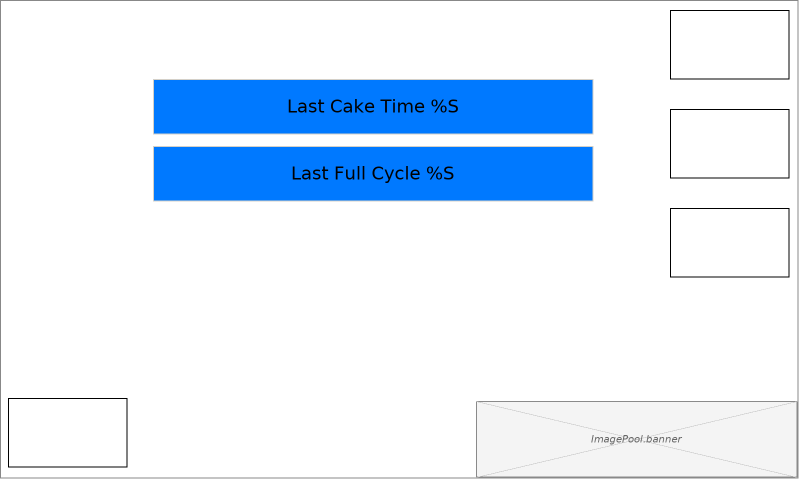
VISUALIZATION Stats  // 799x479, background image ImagePool.background
    Rectangle (670,10 119x69), "SETPOINT"
    Rectangle (670,109 119x69), "MANUAL"
    Rectangle (670,208 119x69), "STATS"
    Rectangle (8,398 119x69), "MAIN"
    Image (476,401 321x76), image: ImagePool.banner
    Label (254,8 266x62), "Stats Screen"
    Textfield (153,79 440x55), "Last Cake Time %S", text variable: GVL_Program_Variables.GVL_CAKE_CYCLE_TIME
    Textfield (153,146 440x55), "Last Full Cycle %S", text variable: GVL_Program_Variables.GVL_FULL_CYCLE_TIME
    hotkey  Id=481040531456, Key=KeyDown=True, KeyName=KEY3_2, ActionToExecute=Action=Assign=Stats, Type=Assignment, VisuElemId=-1
    hotkey  Id=481039482880, Key=KeyDown=True, KeyName=KEY3_3, ActionToExecute=Action=Assign=Manual, Type=Assignment, VisuElemId=-1
    hotkey  Id=481038434304, Key=KeyDown=True, KeyName=KEY3_4, ActionToExecute=Action=Assign=Setpoints, Type=Assignment, VisuElemId=-1
    hotkey  Id=481037385728, Key=KeyDown=True, KeyName=KEY1_5, ActionToExecute=Action=Assign=Main_Screen, Type=Assignment, VisuElemId=-1
END_VISUALIZATION

// CR1082/Application/Pressure_Feed/W77_1
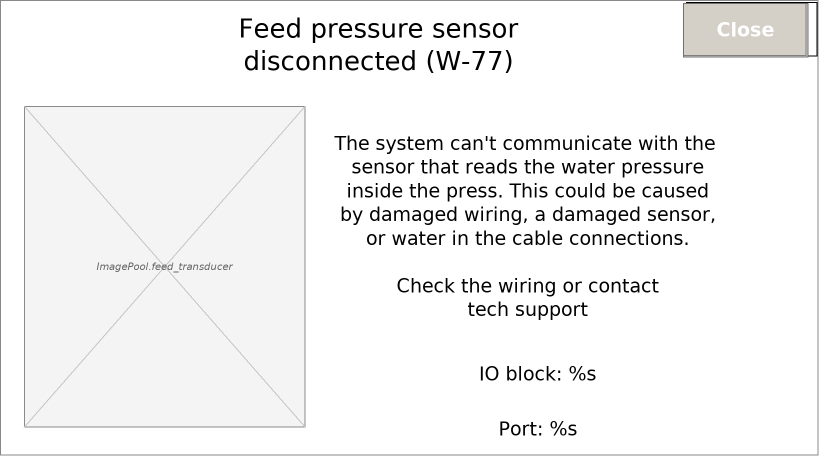
VISUALIZATION W77_1  // 819x456
    Textfield (267,95 522x263), "The system can't communicate with the sensor that reads the water pressure inside the press. This could be caused by damaged wiring, a damaged sensor, or water in the cable connections. Check the wiring or contact tech support", text list: 'TextList_Warnings', text index: 'W_31'
    Textfield (130,6 497x77), "Feed pressure sensor disconnected (W-77)", text list: 'TextList_Warnings', text index: 'W_31_title'
    RoundedRectangle (686,2 131x54)
    Button (683,3 125x54), "Close", text list: 'Button_text', text index: 'Close'
        OnMouseClick: execute {
            IF warnings_globals.warning_screen = 2 THEN
            		VisuElems.CurrentVisu := 'warning_log_2';
            	ELSE
            		VisuElems.CurrentVisu := 'warning_log';
            END_IF
        }
    Textfield (333,349 410x50), "IO block: %s", text variable: pressure_transducer.IO_Link_port.block_name, text list: 'TextList_Warnings', text index: 'W_31'
    Textfield (333,404 410x50), "Port: %s", text variable: pressure_transducer.IO_link_port.port_ID, text list: 'TextList_Warnings', text index: 'W_31'
    Image (24,106 281x321), image: ImagePool.feed_transducer
    hotkey  Id=481081425920, Key=KeyDown=True, KeyName=F5, VisuElemId=57
    hotkey  Id=481082474496, Key=KeyName=F5, VisuElemId=57
END_VISUALIZATION

// CR1082/Application/Pressure_Feed/W78_1
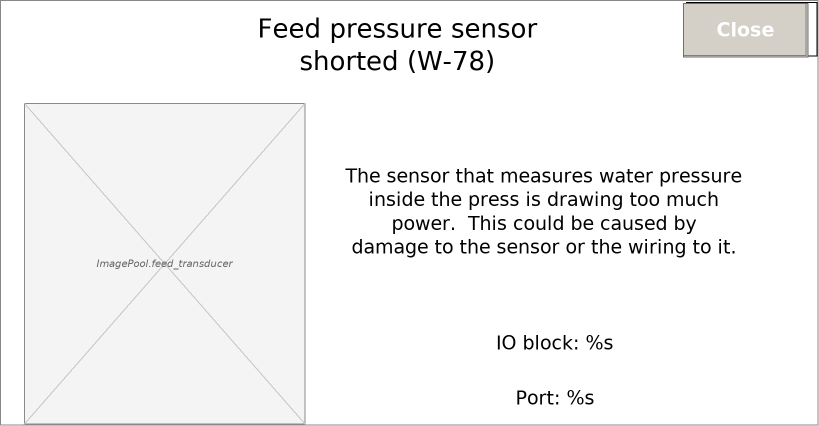
VISUALIZATION W78_1  // 819x426
    Textfield (285,103 518x217), "The sensor that measures water pressure inside the press is drawing too much power. This could be caused by damage to the sensor or the wiring to it.", text list: 'TextList_Warnings', text index: 'W_31'
    Textfield (196,6 403x77), "Feed pressure sensor shorted (W-78)", text list: 'TextList_Warnings', text index: 'W_31_title'
    RoundedRectangle (686,2 131x54)
    Button (683,3 125x54), "Close", text list: 'Button_text', text index: 'Close'
        OnMouseClick: execute {
            IF warnings_globals.warning_screen = 2 THEN
            		VisuElems.CurrentVisu := 'warning_log_2';
            	ELSE
            		VisuElems.CurrentVisu := 'warning_log';
            END_IF
        }
    Textfield (350,318 410x50), "IO block: %s", text variable: pressure_transducer.IO_Link_port.block_name, text list: 'TextList_Warnings', text index: 'W_31'
    Textfield (350,373 410x50), "Port: %s", text variable: pressure_transducer.IO_link_port.port_ID, text list: 'TextList_Warnings', text index: 'W_31'
    Image (24,103 281x321), image: ImagePool.feed_transducer
    hotkey  Id=481081425920, Key=KeyDown=True, KeyName=F5, VisuElemId=57
    hotkey  Id=481082474496, Key=KeyName=F5, VisuElemId=57
END_VISUALIZATION

// CR1082/Application/Pressure_Feed/W79_1
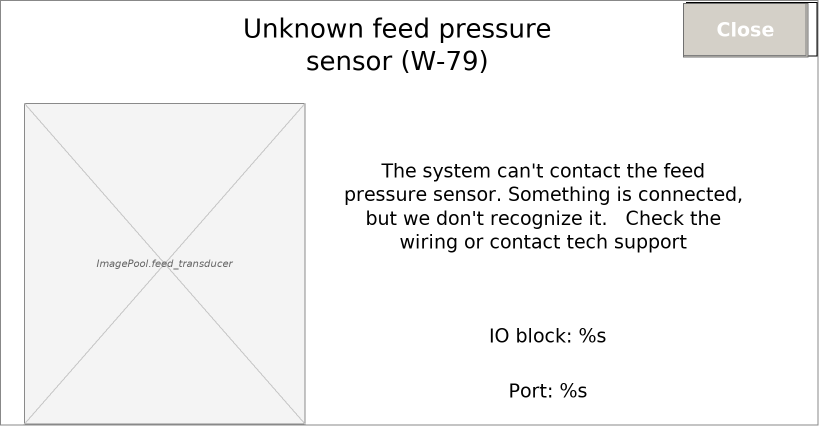
VISUALIZATION W79_1  // 819x426
    Textfield (283,88 521x237), "The system can't contact the feed pressure sensor. Something is connected, but we don't recognize it. Check the wiring or contact tech support", text list: 'TextList_Warnings', text index: 'W_31'
    Textfield (196,6 403x77), "Unknown feed pressure sensor (W-79)", text list: 'TextList_Warnings', text index: 'W_31_title'
    RoundedRectangle (686,2 131x54)
    Button (683,3 125x54), "Close", text list: 'Button_text', text index: 'Close'
        OnMouseClick: execute {
            IF warnings_globals.warning_screen = 2 THEN
            		VisuElems.CurrentVisu := 'warning_log_2';
            	ELSE
            		VisuElems.CurrentVisu := 'warning_log';
            END_IF
        }
    Textfield (343,311 410x50), "IO block: %s", text variable: pressure_transducer.IO_Link_port.block_name, text list: 'TextList_Warnings', text index: 'W_31'
    Textfield (343,366 410x50), "Port: %s", text variable: pressure_transducer.IO_link_port.port_ID, text list: 'TextList_Warnings', text index: 'W_31'
    Image (24,103 281x321), image: ImagePool.feed_transducer
    hotkey  Id=481081425920, Key=KeyDown=True, KeyName=F5, VisuElemId=57
    hotkey  Id=481082474496, Key=KeyName=F5, VisuElemId=57
END_VISUALIZATION

// CR1082/Application/Pressure_Hydraulic/W77
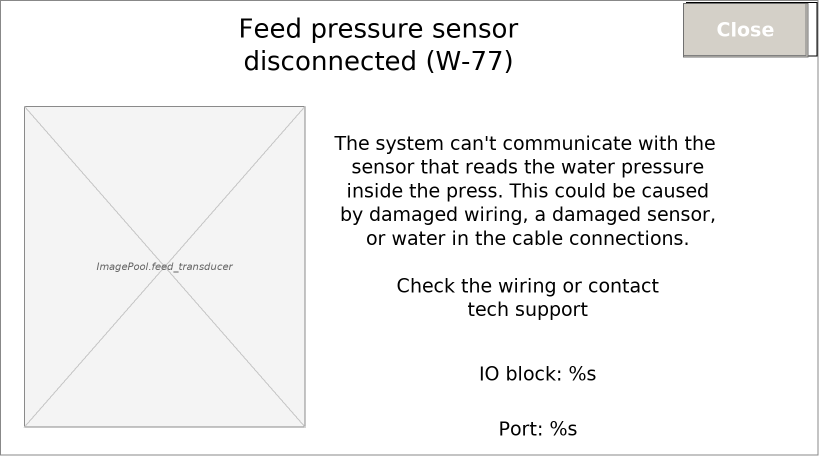
VISUALIZATION W77  // 819x456
    Textfield (267,95 522x263), "The system can't communicate with the sensor that reads the water pressure inside the press. This could be caused by damaged wiring, a damaged sensor, or water in the cable connections. Check the wiring or contact tech support", text list: 'TextList_Warnings', text index: 'W_31'
    Textfield (130,6 497x77), "Feed pressure sensor disconnected (W-77)", text list: 'TextList_Warnings', text index: 'W_31_title'
    RoundedRectangle (686,2 131x54)
    Button (683,3 125x54), "Close", text list: 'Button_text', text index: 'Close'
        OnMouseClick: execute {
            IF warnings_globals.warning_screen = 2 THEN
            		VisuElems.CurrentVisu := 'warning_log_2';
            	ELSE
            		VisuElems.CurrentVisu := 'warning_log';
            END_IF
        }
    Textfield (333,349 410x50), "IO block: %s", text variable: pressure_transducer.IO_Link_port.block_name, text list: 'TextList_Warnings', text index: 'W_31'
    Textfield (333,404 410x50), "Port: %s", text variable: pressure_transducer.IO_link_port.port_ID, text list: 'TextList_Warnings', text index: 'W_31'
    Image (24,106 281x321), image: ImagePool.feed_transducer
    hotkey  Id=481081425920, Key=KeyDown=True, KeyName=F5, VisuElemId=57
    hotkey  Id=481082474496, Key=KeyName=F5, VisuElemId=57
END_VISUALIZATION

// CR1082/Application/Pressure_Hydraulic/W78
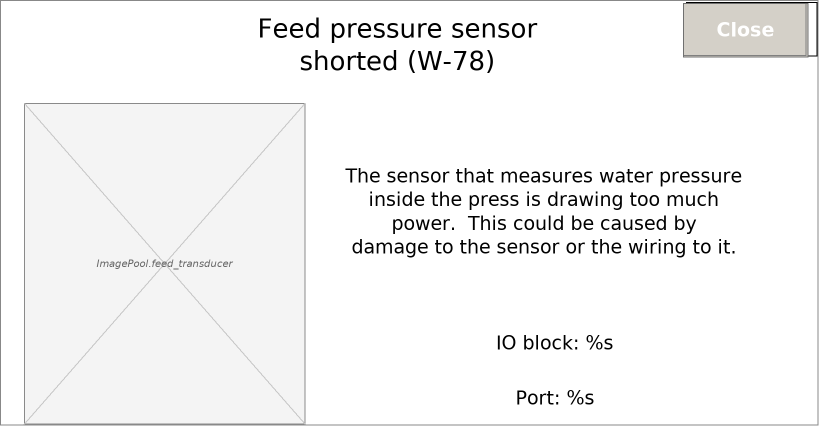
VISUALIZATION W78  // 819x426
    Textfield (285,103 518x217), "The sensor that measures water pressure inside the press is drawing too much power. This could be caused by damage to the sensor or the wiring to it.", text list: 'TextList_Warnings', text index: 'W_31'
    Textfield (196,6 403x77), "Feed pressure sensor shorted (W-78)", text list: 'TextList_Warnings', text index: 'W_31_title'
    RoundedRectangle (686,2 131x54)
    Button (683,3 125x54), "Close", text list: 'Button_text', text index: 'Close'
        OnMouseClick: execute {
            IF warnings_globals.warning_screen = 2 THEN
            		VisuElems.CurrentVisu := 'warning_log_2';
            	ELSE
            		VisuElems.CurrentVisu := 'warning_log';
            END_IF
        }
    Textfield (350,318 410x50), "IO block: %s", text variable: pressure_transducer.IO_Link_port.block_name, text list: 'TextList_Warnings', text index: 'W_31'
    Textfield (350,373 410x50), "Port: %s", text variable: pressure_transducer.IO_link_port.port_ID, text list: 'TextList_Warnings', text index: 'W_31'
    Image (24,103 281x321), image: ImagePool.feed_transducer
    hotkey  Id=481081425920, Key=KeyDown=True, KeyName=F5, VisuElemId=57
    hotkey  Id=481082474496, Key=KeyName=F5, VisuElemId=57
END_VISUALIZATION

// CR1082/Application/Pressure_Hydraulic/W79
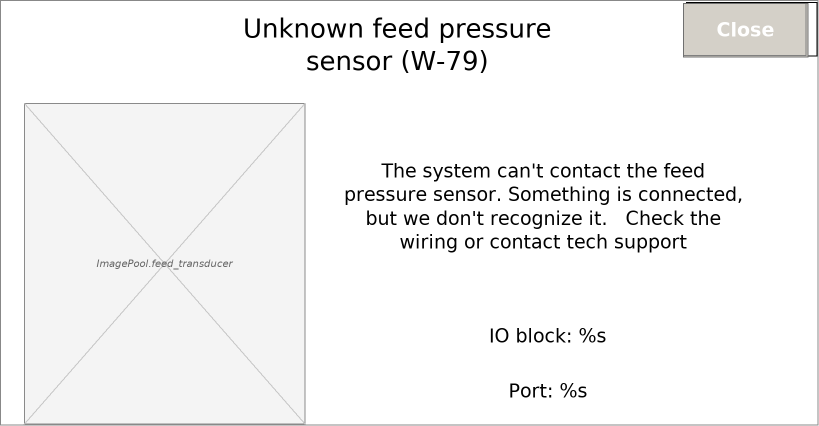
VISUALIZATION W79  // 819x426
    Textfield (283,88 521x237), "The system can't contact the feed pressure sensor. Something is connected, but we don't recognize it. Check the wiring or contact tech support", text list: 'TextList_Warnings', text index: 'W_31'
    Textfield (196,6 403x77), "Unknown feed pressure sensor (W-79)", text list: 'TextList_Warnings', text index: 'W_31_title'
    RoundedRectangle (686,2 131x54)
    Button (683,3 125x54), "Close", text list: 'Button_text', text index: 'Close'
        OnMouseClick: execute {
            IF warnings_globals.warning_screen = 2 THEN
            		VisuElems.CurrentVisu := 'warning_log_2';
            	ELSE
            		VisuElems.CurrentVisu := 'warning_log';
            END_IF
        }
    Textfield (343,311 410x50), "IO block: %s", text variable: pressure_transducer.IO_Link_port.block_name, text list: 'TextList_Warnings', text index: 'W_31'
    Textfield (343,366 410x50), "Port: %s", text variable: pressure_transducer.IO_link_port.port_ID, text list: 'TextList_Warnings', text index: 'W_31'
    Image (24,103 281x321), image: ImagePool.feed_transducer
    hotkey  Id=481081425920, Key=KeyDown=True, KeyName=F5, VisuElemId=57
    hotkey  Id=481082474496, Key=KeyName=F5, VisuElemId=57
END_VISUALIZATION

// CR1082/Application/Warning system/W171
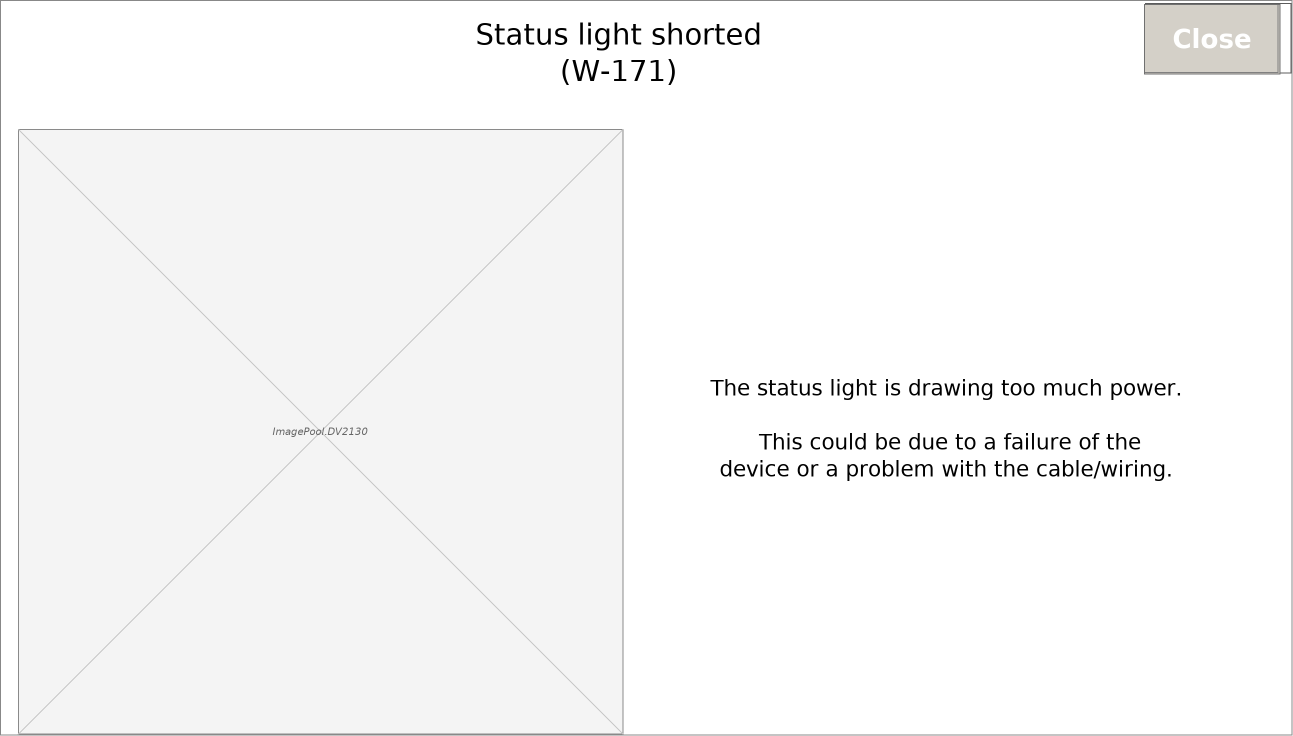
VISUALIZATION W171  // 1293x736
    Textfield (625,254 643x349), "The status light is drawing too much power. This could be due to a failure of the device or a problem with the cable/wiring.", text list: 'TextList_Warnings', text index: 'W_31'
    Textfield (215,13 808x79), "Status light shorted (W-171)", text list: 'TextList_Warnings', text index: 'W_31_title'
    RoundedRectangle (1145,3 146x70)
    Button (1144,4 136x70), "Close", text list: 'Button_text', text index: 'Close'
        OnMouseClick:  Assign=warning_log, Type=Assignment
    Image (18,129 605x605), image: ImagePool.DV2130
    hotkey  Id=481039482880, Key=KeyDown=True, KeyName=F7, VisuElemId=42
    hotkey  Id=481040531456, Key=KeyName=F7, VisuElemId=42
END_VISUALIZATION

// CR1082/Application/Warning system/W172
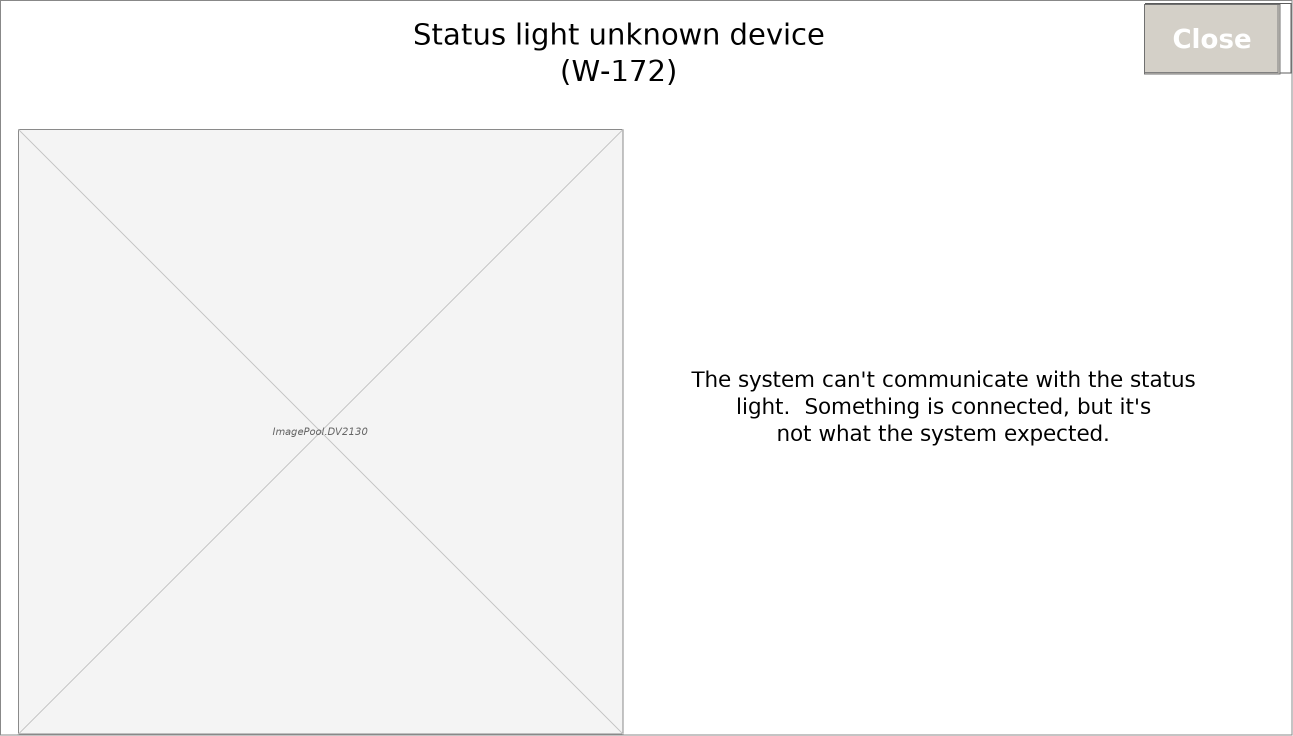
VISUALIZATION W172  // 1293x736
    Image (18,129 605x605), image: ImagePool.DV2130
    Textfield (622,232 643x349), "The system can't communicate with the status light. Something is connected, but it's not what the system expected.", text list: 'TextList_Warnings', text index: 'W_31'
    Textfield (215,13 808x79), "Status light unknown device (W-172)", text list: 'TextList_Warnings', text index: 'W_31_title'
    RoundedRectangle (1145,3 146x70)
    Button (1144,4 136x70), "Close", text list: 'Button_text', text index: 'Close'
        OnMouseClick:  Assign=warning_log, Type=Assignment
    hotkey  Id=481039482880, Key=KeyDown=True, KeyName=F7, VisuElemId=42
    hotkey  Id=481040531456, Key=KeyName=F7, VisuElemId=42
END_VISUALIZATION

// CR1082/Application/Warning system/W25
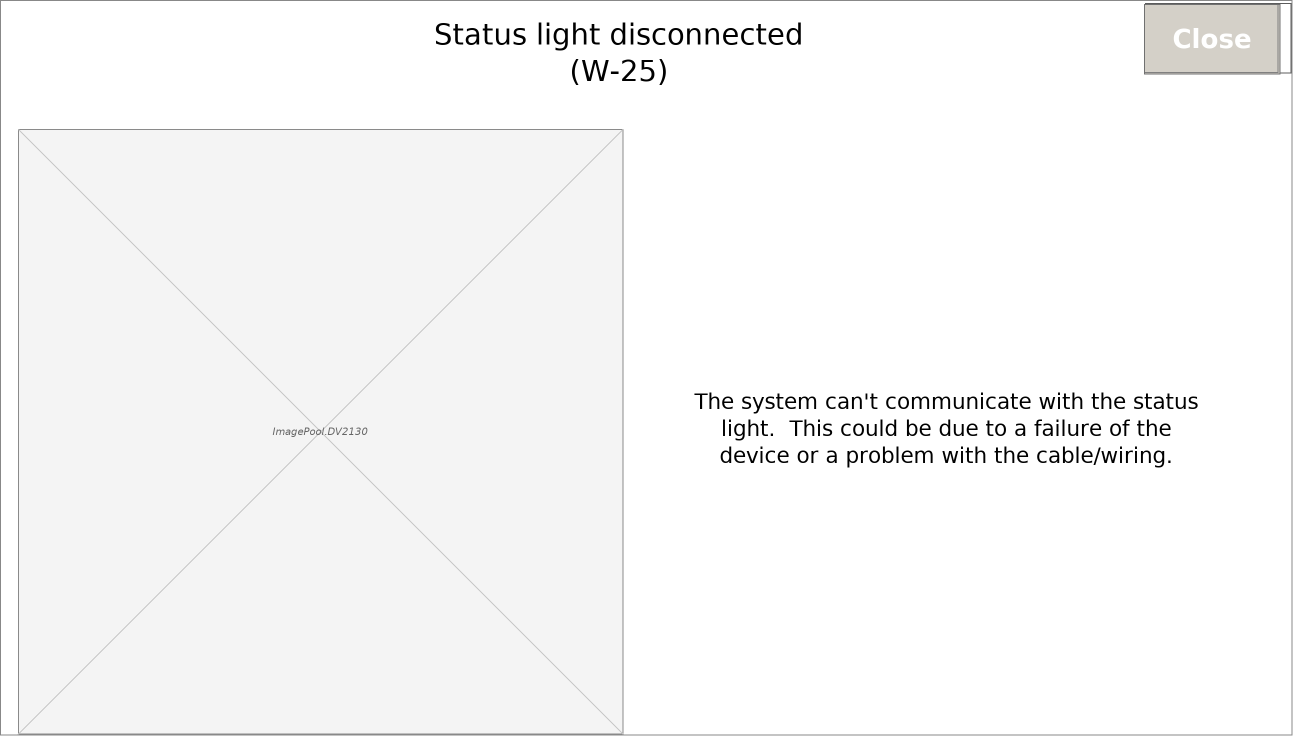
VISUALIZATION W25  // 1293x736
    Textfield (625,254 643x349), "The system can't communicate with the status light. This could be due to a failure of the device or a problem with the cable/wiring.", text list: 'TextList_Warnings', text index: 'W_31'
    Textfield (215,13 808x79), "Status light disconnected (W-25)", text list: 'TextList_Warnings', text index: 'W_31_title'
    RoundedRectangle (1145,3 146x70)
    Button (1144,4 136x70), "Close", text list: 'Button_text', text index: 'Close'
        OnMouseClick:  Assign=warning_log, Type=Assignment
    Image (18,129 605x605), image: ImagePool.DV2130
    hotkey  Id=481039482880, Key=KeyDown=True, KeyName=F7, VisuElemId=42
    hotkey  Id=481040531456, Key=KeyName=F7, VisuElemId=42
END_VISUALIZATION

// CR1082/Application/Warning system/W97
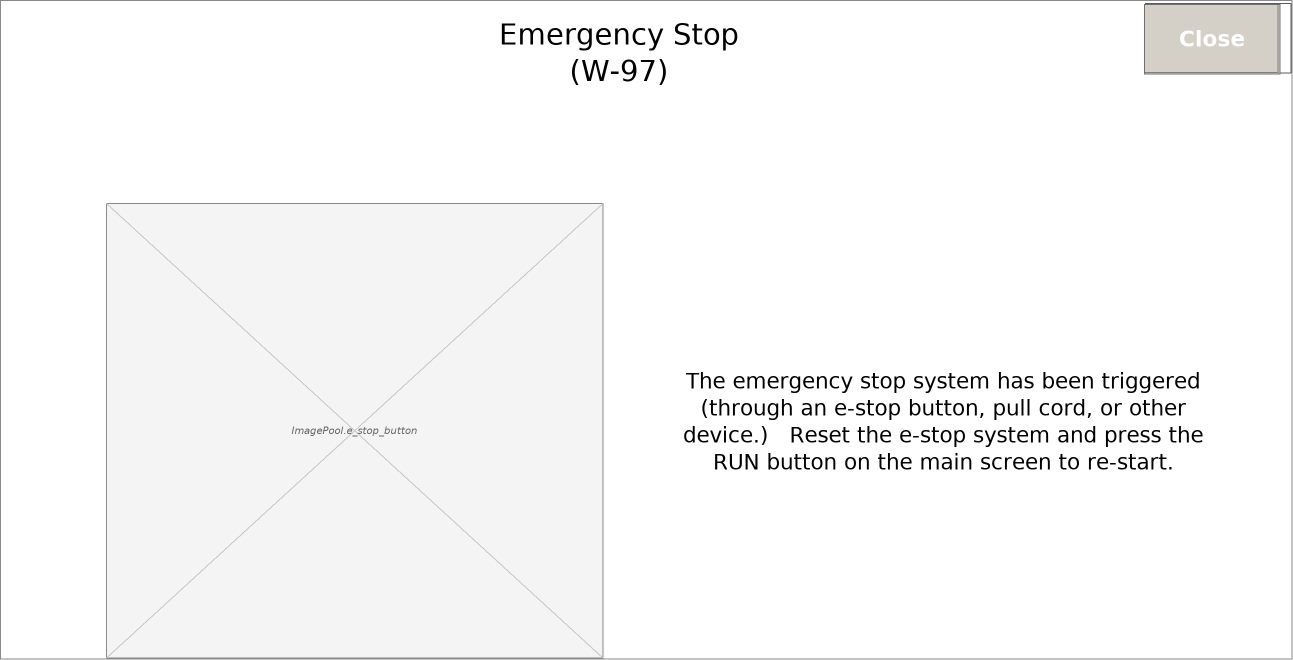
VISUALIZATION W97  // 1293x660
    Textfield (607,247 673x349), "The emergency stop system has been triggered (through an e-stop button, pull cord, or other device.) Reset the e-stop system and press the RUN button on the main screen to re-start.", text list: 'TextList_Warnings', text index: 'W_31'
    Textfield (215,13 808x79), "Emergency Stop (W-97)", text list: 'TextList_Warnings', text index: 'W_31_title'
    RoundedRectangle (1145,3 146x70)
    Button (1144,4 136x70), "Close", text list: 'Button_text', text index: 'Close'
        OnMouseClick:  Assign=warning_log, Type=Assignment
    Image (106,203 497x455), image: ImagePool.e_stop_button
    hotkey  Id=481039482880, Key=KeyDown=True, KeyName=F7, VisuElemId=42
    hotkey  Id=481040531456, Key=KeyName=F7, VisuElemId=42
END_VISUALIZATION

// ecomatDisplay43inch_64bit/Application/Pressure_Feed/W77_1
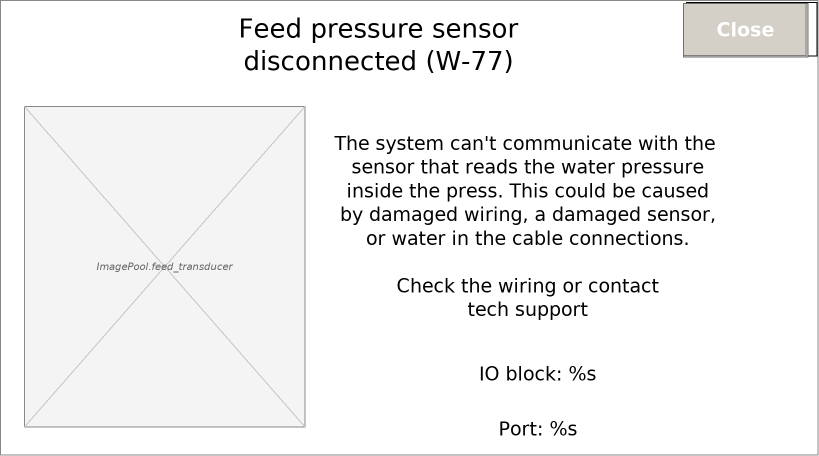
VISUALIZATION W77_1  // 819x456
    Textfield (267,95 522x263), "The system can't communicate with the sensor that reads the water pressure inside the press. This could be caused by damaged wiring, a damaged sensor, or water in the cable connections. Check the wiring or contact tech support", text list: 'TextList_Warnings', text index: 'W_31'
    Textfield (130,6 497x77), "Feed pressure sensor disconnected (W-77)", text list: 'TextList_Warnings', text index: 'W_31_title'
    RoundedRectangle (686,2 131x54)
    Button (683,3 125x54), "Close", text list: 'Button_text', text index: 'Close'
        OnMouseClick: execute {
            IF warnings_globals.warning_screen = 2 THEN
            		VisuElems.CurrentVisu := 'warning_log_2';
            	ELSE
            		VisuElems.CurrentVisu := 'warning_log';
            END_IF
        }
    Textfield (333,349 410x50), "IO block: %s", text variable: pressure_transducer.IO_Link_port.block_name, text list: 'TextList_Warnings', text index: 'W_31'
    Textfield (333,404 410x50), "Port: %s", text variable: pressure_transducer.IO_link_port.port_ID, text list: 'TextList_Warnings', text index: 'W_31'
    Image (24,106 281x321), image: ImagePool.feed_transducer
    hotkey  Id=481081425920, Key=KeyDown=True, KeyName=F5, VisuElemId=57
    hotkey  Id=481082474496, Key=KeyName=F5, VisuElemId=57
END_VISUALIZATION

// ecomatDisplay43inch_64bit/Application/Pressure_Feed/W78_1
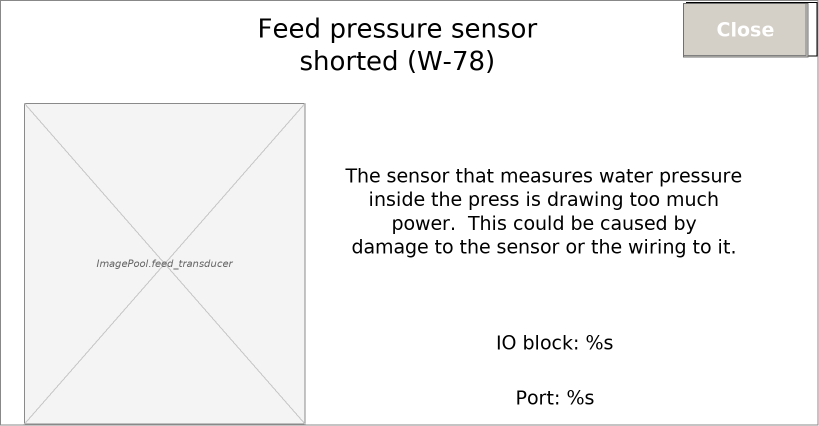
VISUALIZATION W78_1  // 819x426
    Textfield (285,103 518x217), "The sensor that measures water pressure inside the press is drawing too much power. This could be caused by damage to the sensor or the wiring to it.", text list: 'TextList_Warnings', text index: 'W_31'
    Textfield (196,6 403x77), "Feed pressure sensor shorted (W-78)", text list: 'TextList_Warnings', text index: 'W_31_title'
    RoundedRectangle (686,2 131x54)
    Button (683,3 125x54), "Close", text list: 'Button_text', text index: 'Close'
        OnMouseClick: execute {
            IF warnings_globals.warning_screen = 2 THEN
            		VisuElems.CurrentVisu := 'warning_log_2';
            	ELSE
            		VisuElems.CurrentVisu := 'warning_log';
            END_IF
        }
    Textfield (350,318 410x50), "IO block: %s", text variable: pressure_transducer.IO_Link_port.block_name, text list: 'TextList_Warnings', text index: 'W_31'
    Textfield (350,373 410x50), "Port: %s", text variable: pressure_transducer.IO_link_port.port_ID, text list: 'TextList_Warnings', text index: 'W_31'
    Image (24,103 281x321), image: ImagePool.feed_transducer
    hotkey  Id=481081425920, Key=KeyDown=True, KeyName=F5, VisuElemId=57
    hotkey  Id=481082474496, Key=KeyName=F5, VisuElemId=57
END_VISUALIZATION
